(*----------------------------------------------------------------------------------------------------------------------------------------*)
(*Invoke Large Type Services Stand (Pnuematic I/O)*)
(*----------------------------------------------------------------------------------------------------------------------------------------*)
	(*Input Data*)
	SS01.Prev_EcatNode_Present:= NOT IS01.EK1100_NotPresent; (*Ensure Previous Node Exists to determine Ecat Cable Break of this Devices Input Cable*)
	SS01.Output_Req.0:= All_Estops_OK AND GTAC_CONFIG.Option_Air1; (*air valve 1*)
	SS01.Output_Req.1:= All_Estops_OK AND GTAC_CONFIG.Option_Air1; (*air valve 2*)
	SS01.Output_REQ.2:= RollDoor01.DoorClose_CMD;
	SS01.Output_REQ.3:= RollDoor01.DoorOpen_CMD;
	SS01.Output_REQ.4:= FALSE;
	SS01.Output_REQ.5:= FALSE;
	SS01.Output_REQ.6:= FALSE;
	SS01.Output_REQ.7:= FALSE;
	SS01.FB_In.Option_EP9214_Count:= GTAC_CONFIG.Option_EP9214_Count;
	(*Call Actual Function*)
	SS01();
	(*Output Data*)
	Out_To_ICxx.SS[1].Discrete_Image:= SS01.Discrete_Image;
	Out_To_ICxx.SS[1].ECAT_Cable_Breaks:= SS01.EcatSlave_Cable_Breaks;

	(*Input Data*)
	(*SS02.Prev_EcatNode_Present:= NOT SS01.EP1008_NotPresent; (*Ensure Previous Node Exists to determine Ecat Cable Break of this Devices Input Cable*)
	SS02.Output_Req.0:= All_Estops_OK AND GTAC_CONFIG.Option_Air2; (*air valve 1*)
	SS02.Output_Req.1:= All_Estops_OK AND GTAC_CONFIG.Option_Air2; (*air valve 2*)
	SS02.Output_REQ.2:= FALSE;
	SS02.Output_REQ.3:= FALSE;
	SS02.Output_REQ.4:= FALSE;
	SS02.Output_REQ.5:= FALSE;
	SS02.Output_REQ.6:= FALSE;
	SS02.Output_REQ.7:= FALSE;
	(*Call Actual Function*)
	SS02();
	(*Output Data*)
	Out_To_ICxx.SS[2].Discrete_Image:= SS02.Discrete_Image;
	Out_To_ICxx.SS[2].ECAT_Cable_Breaks:= SS02.EcatSlave_Cable_Breaks;*)


(*----------------------------------------------------------------------------------------------------------------------------------------*)
(* Invoke Enabling Swtich Plates*)
(*----------------------------------------------------------------------------------------------------------------------------------------*)
	(*Input Data*)
	ESW01.Prev_EcatNode_Present:= NOT MAIN.R3.EL6695_PortC_MissingLink; (*Ensure Previous Node Exists to determine Ecat Cable Break of this Devices Input Cable*)
	(*Call Actual Function*)
	ESW01();
	(*Output Data*)
	Out_To_ICxx.ESW[1].Discrete_Image:= ESW01.Discrete_Image;
	Out_To_ICxx.ESW[1].ECAT_Cable_Breaks:= ESW01.EcatSlave_Cable_Breaks;
	
	(*Input Data*)
	ESW02.Prev_EcatNode_Present:= NOT MAIN.IC03.EK1100_NotPresent; (*Ensure Previous Node Exists to determine Ecat Cable Break of this Devices Input Cable*)
	(*Call Actual Function*)
	ESW02();
	(*Output Data*)
	Out_To_ICxx.ESW[2].Discrete_Image:= ESW02.Discrete_Image;
	Out_To_ICxx.ESW[2].ECAT_Cable_Breaks:= ESW02.EcatSlave_Cable_Breaks;

	(*Input Data*)
	ESW03.Prev_EcatNode_Present:= NOT MAIN.IC02.EK1100_NotPresent; (*Ensure Previous Node Exists to determine Ecat Cable Break of this Devices Input Cable*)
	(*Call Actual Function*)
	ESW03();
	(*Output Data*)
	Out_To_ICxx.ESW[3].Discrete_Image:= ESW03.Discrete_Image;
	Out_To_ICxx.ESW[3].ECAT_Cable_Breaks:= ESW03.EcatSlave_Cable_Breaks;

(*----------------------------------------------------------------------------------------------------------------------------------------*)
(*Invoke EOAT FBs and Subordinate Fixtures*)
(*----------------------------------------------------------------------------------------------------------------------------------------*)
	(*EOATs Action*)
	EOATs();

(*----------------------------------------------------------------------------------------------------------------------------------------*)
(*Invoke IC FBs and Subordinate Fixtures*)
(*----------------------------------------------------------------------------------------------------------------------------------------*)
	(*ICs Action*)
	ICs();
	
(*----------------------------------------------------------------------------------------------------------------------------------------*)
(*Invoke Product Tracking Action*)
(*----------------------------------------------------------------------------------------------------------------------------------------*)
	(*Product Tracking Action*)
	Product_Tracking();

(*-------------------------------------------------------------------------------------------------------------------------------------*)
(*Invoke Robot FBs*)
(*-------------------------------------------------------------------------------------------------------------------------------------*)
	(*Robots Action*)
	Robots();

	
(*-------------------------------------------------------------------------------------------------------------------------------------*)
(*-------------------------------------------------------------------------------------------------------------------------------------*)
(*---------------------------------------------------- End of MAIN---------------------------------------------------------------------*)
(*-------------------------------------------------------------------------------------------------------------------------------------*)
(*-------------------------------------------------------------------------------------------------------------------------------------*)

ACTION EOATs:



	(*R04 - EOAT 04*)
		EOAT04(

			Enable_Motion:= R4.Servos_Are_On,
			Dry_Cycle:= GTAC_CONFIG.Dry_Cycle_Enabled,
			Robot_WorkingOK:= ((R4.Task_ID_Ack=PickUP_Fix01) OR (R4.Task_ID_Ack=Work_PED01)) AND R4.Operating,

			(*Set Configuration Data Here*)
			ID:= 4,							(*Set EOAT ID*)
			NodeLayout:= Main.ECAT_Master.EOATNodeLayout[4],	(*Pass in Assembled Node layout for UI*)
			Input_Node_Count:= 5,				(*Set Expected Input Node Count(Current Limit is 9*)
			VB_Node_Count:= 1,				(*Set Expected Input Node Count(Current Limit is 3*)
	
			(*Input Data*)
			(*Use Command All Sensors if your gripper has common part for the entire gripper.*)
			(*Use Command Sensors Group1/Group 2 if your gripper has multiple parts for the entire gripper. EX: LH and RH part*)
			CMD_CheckAllSensors_OFF:= FALSE, 
			CMD_CheckSensorsOFF_Grp1:= R4.EOAT_Req.0, (*129*) (*Sensors 1-2*)
			CMD_CheckSensorsOFF_Grp2:= R4.EOAT_Req.2, (*131*) (*Sensors 3-4*)
			CMD_CheckSensorsOFF_Grp3:= FALSE,
			CMD_CheckSensorsOFF_Grp4:= FALSE,
			CMD_CheckSensorsOFF_Grp5:= FALSE,

			CMD_CheckAllSensors_ON:= FALSE,
			CMD_CheckSensorsON_Grp1:= R4.EOAT_Req.1, (*130*) (*Sensors 1-2*)
			CMD_CheckSensorsON_Grp2:= R4.EOAT_Req.3, (*132*) (*Sensors 3-4*)
			CMD_CheckSensorsON_Grp3:= FALSE,
			CMD_CheckSensorsON_Grp4:= FALSE,
			CMD_CheckSensorsON_Grp5:= FALSE,

			(*Use Command Tool to Work/HOME if your gripper has common part for the entire gripper.*)
			(*Use Clamps Groups if your gripper has a LH/RH part for the gripper.*)
			CMD_Tool_To_WORK:= FALSE,
			CMD_CylToWORK_Grp1:= R4.EOAT_Req.4, (*133*) (*Clamps 1-4*)
			CMD_CylToWORK_Grp2:= R4.EOAT_Req.6, (*135*) (*Clamps 5-8*)
			CMD_CylToWORK_Grp3:= R4.EOAT_Req.8, (*137*) (*Pins 1-2*)
			CMD_CylToWORK_Grp4:= R4.EOAT_Req.10, (*139*) (*Pins 3-4*)
			CMD_CylToWORK_Grp5:= FALSE,

			CMD_Tool_To_HOME:= FALSE,
			CMD_CylToHOME_Grp1:= R4.EOAT_Req.5, (*134*) (*Clamps 1-4*)
			CMD_CylToHOME_Grp2:= R4.EOAT_Req.7, (*136*) (*Clamps 5-8*)
			CMD_CylToHOME_Grp3:= R4.EOAT_Req.9, (*138*) (*Pins 1-2*)
			CMD_CylToHOME_Grp4:= R4.EOAT_Req.11, (*140*) (*Pins 3-4*)
			CMD_CylToHOME_Grp5:= FALSE
			);
		(*Output Data*)
		Out_To_ICxx.EOAT04_Discrete_Image:= EOAT04.Discrete_Image;
		Out_To_ICxx.ProductReport[34]:= EOAT04_1_ProductData_Pers; 	(*Transfer Product Data to UI*)
		Out_To_ICxx.ProductReport[35]:= EOAT04_2_ProductData_Pers; 	(*Transfer Product Data to UI*)

		(*Output Data - Send ACKs bak to Robot*)
		(*Sensor ACKs*)
		R4.FB_In.EOATReq_Ack.0:= EOAT04.EOAT_Part1_Empty;	(*129*) //R4.EOAT_Req.0 AND DEBUG - removed to make more automated. delete if tested good
		R4.FB_In.EOATReq_Ack.1:= EOAT04.Part1_In_EOAT;		(*130*) //R4.EOAT_Req.1 AND DEBUG
		R4.FB_In.EOATReq_Ack.2:= EOAT04.EOAT_Part2_Empty;	(*131*) //R4.EOAT_Req.2 AND DEBUG 
		R4.FB_In.EOATReq_Ack.3:= EOAT04.Part2_In_EOAT;		(*132*) //R4.EOAT_Req.3 AND DEBUG
		
		(*CLAMP ACKs*)
		R4.FB_In.EOATReq_Ack.4:= R4.EOAT_Req.4 AND EOAT04.ACK_CylAtWORK_Grp1;	(*133*)
		R4.FB_In.EOATReq_Ack.5:= R4.EOAT_Req.5 AND EOAT04.ACK_CylAtHOME_Grp1;	(*134*)		
		R4.FB_In.EOATReq_Ack.6:= R4.EOAT_Req.6 AND EOAT04.ACK_CylAtWORK_Grp2;	(*135*)
		R4.FB_In.EOATReq_Ack.7:= R4.EOAT_Req.7 AND EOAT04.ACK_CylAtHOME_Grp2;	(*136*)
		
		(*Pin ACKs*)
		R4.FB_In.EOATReq_Ack.8:= R4.EOAT_Req.8 AND EOAT04.ACK_CylAtWORK_Grp3;	(*137*)
		R4.FB_In.EOATReq_Ack.9:= R4.EOAT_Req.9 AND EOAT04.ACK_CylAtHOME_Grp3;	(*138*)		
		R4.FB_In.EOATReq_Ack.10:= R4.EOAT_Req.10 AND EOAT04.ACK_CylAtWORK_Grp4;	(*139*)
		R4.FB_In.EOATReq_Ack.11:= R4.EOAT_Req.11 AND EOAT04.ACK_CylAtHOME_Grp4;	(*140*)

	(*Additional EOAT can be added here. Up to 30*)
	(*Please update the faults if you add additional EOAT*)
END_ACTION

ACTION ICs:



	(*Industrial Controller 01*)
	(*Input Data*)
	IC01.FB_In.Safety_RST:=SAFETY_RESET;
	IC01.FB_In.Enable_Motion:= All_Estops_OK AND All_SafetyGates_OK;
	IC01.FB_In.Estops_OK:= All_Estops_OK;
	IC01.FB_In.Safety_Gates_Ok:= All_SafetyGates_OK;
	IC01.FB_In.CoE_Read_Trigger:= (GTAC_CONFIG.Option_IC_Count>=1) AND Pulse_CoERead;	(*Global Interval of CoE Reads*)
	IC01.FB_In.Ecat_Master_AmsNetID:= MAIN.ECAT_Master.AmsID;
	IC01.FB_In.Prev_EcatNode_Present:= TRUE; 												(*Ensure Previous Node Exists to determine Ecat Cable Break of this Devices Input Cable*)
	IC01.FB_In.Output_Req1:= In_From_ICxx.LockSGK1;
	IC01.Turntable_Type:= TRUE;	(*Debug - Set to true if using a turntable. this will change the status light based on table position. set to false if no turntable.*)
	IC01.Op1_At_Operator:= Fix01.TurntableB_At_Robot OR (MAIN.R1.Task_ID_Ack=Sweep_Fix01) OR (MAIN.R2.Task_ID_Ack=Sweep_Fix01) OR (MAIN.R1.Task_ID_Ack=Sweep_Fix02) OR (MAIN.R2.Task_ID_Ack=Sweep_Fix02);
	IC01.Op2_At_Operator:= Fix01.TurntableA_At_Robot OR (MAIN.R1.Task_ID_Ack=Sweep_Fix01) OR (MAIN.R2.Task_ID_Ack=Sweep_Fix01) OR (MAIN.R1.Task_ID_Ack=Sweep_Fix02) OR (MAIN.R2.Task_ID_Ack=Sweep_Fix02);
	IC01.FB_In.OP1_Green_LampReq:= Fix01.Ready_To_Load;
	IC01.FB_In.OP2_Green_LampReq:= Fix03.Ready_To_Load;
	IC01.FB_In.OP1_Yellow_LampReq:= TRUE;
	IC01.FB_In.OP2_Yellow_LampReq:= TRUE;
	IC01.FB_In.OP1_Red_LampReq:= Fix01.Red_Lamp_Req OR Faults.System_Major_Fault;
	IC01.FB_In.OP2_Red_LampReq:= Fix03.Red_Lamp_Req OR Faults.System_Major_Fault;
	IC01.OP1_LC_Clear:= IC01.OP1_HumanVertLC_Clear AND IC01.OP1_HumanHorizLC_Clear AND IC01.OP1_RobotVertLC_Clear AND IC01.OP2_HumanVertLC_Clear AND IC01.OP2_HumanHorizLC_Clear;
	IC01.OP2_LC_Clear:= IC01.OP1_HumanVertLC_Clear AND IC01.OP1_HumanHorizLC_Clear AND IC01.OP1_RobotVertLC_Clear AND IC01.OP2_HumanVertLC_Clear AND IC01.OP2_HumanHorizLC_Clear;
	(*Call FUNCTION*)
	IC01();
	(*Output IC Data to All ICs*)
	Out_To_ICxx.IC[1].Discrete_Image:= IC01.Discrete_Image;
	Out_To_ICxx.IC[1].ECAT_Cable_Breaks:= IC01.ECatSlave_Cable_Breaks;
	Out_To_ICxx.IC01OP1_LCHVR:= IC01.OP1_HumanVertLC_Clear;
	Out_To_ICxx.IC01OP1_LCHHR:= IC01.OP1_HumanHorizLC_Clear;
	Out_To_ICxx.IC01OP1_LCRVR:= IC01.OP1_RobotVertLC_Clear; (*DEBUG - ADD OR REMOVE TO OTHER LIGHT CURTAINS. BYPASSES INDICATOR ON UI*)
	Out_To_ICxx.IC01OP2_LCHVR:= IC01.OP2_HumanVertLC_Clear;
	Out_To_ICxx.IC01OP2_LCHHR:= IC01.OP2_HumanHorizLC_Clear;
	Out_To_ICxx.IC01OP2_LCRVR:= IC01.OP2_RobotVertLC_Clear;
	
		(*OP1*)
			(*Fixture 01*)
			(*Input Data*)
			Fix01.Enable_Motion:= IC01.OP1_Enable_Motion;
			Fix01.Discrete_In:= In_From_ICxx.Fix01_Discrete_In;
			Fix01.Discrete_In.ModelData:= In_From_ICxx.Fix01_Discrete_In.ModelData;
			Fix01.NodeLayout:= Main.ECAT_Master.FixNodeLayout[1];				(*Pass in Assembled Node layout for UI*)
			Fix01.Discrete_In.Input_Node_Count:= 29;								(*Overridden for now, later version will map from UI read config sheet*)
			Fix01.Discrete_In.VB_Node_Count:= 2;								(*Overridden for now, later version will map from UI read config sheet*)
			Fix01.Discrete_In.Output_Node_Count:= 0;								(*Overridden for now, later version will map from UI read config sheet*)
			Fix01.Discrete_In.Water_Stand_Count:= 0;							(*Overridden for now, later version will map from UI read config sheet*)
			Fix01.Dry_Cycle:= GTAC_CONFIG.Dry_Cycle_Enabled OR GTAC_CONFIG.Local_DryCycle_Enables.1;
			Fix01.Cell_In_Services:= Cell_Services_Prog.Service_Call_ForAllRobots OR In_From_ICxx.Cycle_Hold;
			Fix01.Flash_Rate:= Pulse_1S;

			(*Call FUNCTION*)
			Fix01();
			(*Output Data*)
			Out_To_ICxx.Fix01_Discrete_Image:= Fix01.Discrete_Image;

		
			(*Fixture 02*)
			(*Input Data*)
			Fix02.Enable_Motion:= IC01.OP2_Enable_Motion;
			Fix02.Discrete_In:= In_From_ICxx.Fix02_Discrete_In;
			Fix02.Discrete_In.ModelData:= In_From_ICxx.Fix02_Discrete_In.ModelData;
			Fix02.NodeLayout:= Main.ECAT_Master.FixNodeLayout[2];				(*Pass in Assembled Node layout for UI*)
			Fix02.Discrete_In.Input_Node_Count:= 29;								(*Overridden for now, later version will map from UI read config sheet*)
			Fix02.Discrete_In.VB_Node_Count:= 2;								(*Overridden for now, later version will map from UI read config sheet*)
			Fix02.Discrete_In.Output_Node_Count:= 0;								(*Overridden for now, later version will map from UI read config sheet*)
			Fix02.Discrete_In.Water_Stand_Count:= 0;								(*Overridden for now, later version will map from UI read config sheet*)
			Fix02.Dry_Cycle:= GTAC_CONFIG.Dry_Cycle_Enabled OR GTAC_CONFIG.Local_DryCycle_Enables.2;
			Fix02.Cell_In_Services:= Cell_Services_Prog.Service_Call_ForAllRobots OR In_From_ICxx.Cycle_Hold;
			Fix02.Flash_Rate:= Pulse_1S;
			(*Call FUNCTION*)
			Fix02();
			(*Output Data*)
			Out_To_ICxx.Fix02_Discrete_Image:= Fix02.Discrete_Image;

	(*Industrial Controller 02*)
	(*Input Data*)
	IC02.FB_In.Safety_RST:=SAFETY_RESET;
	IC02.FB_In.Enable_Motion:= All_Estops_OK AND All_SafetyGates_OK;
	IC02.FB_In.Estops_OK:= All_Estops_OK;
	IC02.FB_In.Safety_Gates_Ok:= All_SafetyGates_OK;
	IC02.FB_In.CoE_Read_Trigger:= (GTAC_CONFIG.Option_IC_Count>=2) AND Pulse_CoERead;	(*Global Interval of CoE Reads*)
	IC02.FB_In.Ecat_Master_AmsNetID:= MAIN.ECAT_Master.AmsID;
	IC02.FB_In.Prev_EcatNode_Present:= NOT MAIN.MD02.EP2624_PortB_MissingLink ; 						(*Ensure Previous Node Exists to determine Ecat Cable Break of this Devices Input Cable*)
	IC02.FB_In.Output_Req1:= In_From_ICxx.LockSGK1 OR In_From_ICxx.LockSGK2;
	IC02.Turntable_Type:= TRUE;	(*Debug - Set to true if using a turntable. this will change the status light based on table position. set to false if no turntable.*)
	IC02.Op1_At_Operator:= Fix03.TurntableB_At_Robot OR (MAIN.R3.Task_ID_Ack=Sweep_Fix03) OR (MAIN.R4.Task_ID_Ack=Sweep_Fix03) OR (MAIN.R3.Task_ID_Ack=Sweep_Fix04) OR (MAIN.R4.Task_ID_Ack=Sweep_Fix04); (*debug - change robot*)
	IC02.Op2_At_Operator:= Fix03.TurntableA_At_Robot OR (MAIN.R3.Task_ID_Ack=Sweep_Fix03) OR (MAIN.R4.Task_ID_Ack=Sweep_Fix03) OR (MAIN.R3.Task_ID_Ack=Sweep_Fix04) OR (MAIN.R4.Task_ID_Ack=Sweep_Fix04); (*debug - change robot*)
	IC02.FB_In.OP1_Green_LampReq:= Fix03.Ready_To_Load;
	IC02.FB_In.OP2_Green_LampReq:= Fix04.Ready_To_Load;
	IC02.FB_In.OP1_Yellow_LampReq:= TRUE;
	IC02.FB_In.OP2_Yellow_LampReq:= TRUE;
	IC02.FB_In.OP1_Red_LampReq:= Fix03.Red_Lamp_Req OR Faults.System_Major_Fault;
	IC02.FB_In.OP2_Red_LampReq:= Fix04.Red_Lamp_Req OR Faults.System_Major_Fault;
	IC02.OP1_LC_Clear:= IC02.OP1_HumanVertLC_Clear AND IC02.OP1_HumanHorizLC_Clear AND IC02.OP1_RobotVertLC_Clear AND IC02.OP2_HumanVertLC_Clear AND IC02.OP2_HumanHorizLC_Clear;
	IC02.OP2_LC_Clear:= IC02.OP1_HumanVertLC_Clear AND IC02.OP1_HumanHorizLC_Clear AND IC02.OP1_RobotVertLC_Clear AND IC02.OP2_HumanVertLC_Clear AND IC02.OP2_HumanHorizLC_Clear;
	(*Call FUNCTION*)
	IC02();
	(*Output IC Data to all ICs*)
	Out_To_ICxx.IC[2].Discrete_Image:= IC02.Discrete_Image;
	Out_To_ICxx.IC[2].ECAT_Cable_Breaks:= IC02.ECatSlave_Cable_Breaks;
	Out_To_ICxx.IC02OP1_LCHVR:= IC02.OP1_HumanVertLC_Clear;
	Out_To_ICxx.IC02OP1_LCHHR:= IC02.OP1_HumanHorizLC_Clear;
	Out_To_ICxx.IC02OP1_LCRVR:= IC02.OP1_RobotVertLC_Clear;
	Out_To_ICxx.IC02OP2_LCHVR:= IC02.OP2_HumanVertLC_Clear;
	Out_To_ICxx.IC02OP2_LCHHR:= IC02.OP2_HumanHorizLC_Clear;
	Out_To_ICxx.IC02OP2_LCRVR:= IC02.OP2_RobotVertLC_Clear;

		(*OP1*)
			(*Fixture 03*)
			(*Input Data*)
			Fix03.Enable_Motion:= IC02.OP1_Enable_Motion;
			Fix03.Discrete_In:= In_From_ICxx.Fix03_Discrete_In;
			(*Perform Look ahead for Model data depending on line loading*)
			
				(*Valid part For this Fix in EOAT04_1, so use EOAT_1 model*)
				IF ((EOAT04.Part1_In_EOAT AND NOT Fix03.Load_Complete) OR Fix03.Repo_REQS.0) AND Fix03.Part_InEOAT04_1_ReadyforThisFix 
					THEN
					Fix03.Discrete_In.ModelData:= EOAT04_1_ProductData_Pers.Product_Model_ID;
	
				(*Valid part For this Fix in EOAT04_2, so use EOAT_2 model*)
				ELSIF ((EOAT04.Part2_In_EOAT AND NOT Fix03.Load_Complete) OR Fix03.Repo_REQS.0) AND Fix03.Part_InEOAT04_2_ReadyforThisFix
					THEN
					Fix03.Discrete_In.ModelData:= EOAT04_2_ProductData_Pers.Product_Model_ID;
	
				(*No valid part in EOAT04, but valid part in Fix101, so use Fix101 model*)
				ELSIF (((NOT Fix03.Load_Complete OR Fix03.Unload_Complete) AND Fix101.Load_Complete) OR (MAIN.R4.Task_ID_Ack = PickUp_Fix101)) AND 
						NOT Fix03.Part_InEOAT04_1_ReadyforThisFix AND NOT Fix03.Part_InEOAT04_2_ReadyforThisFix AND (MAIN.R4.Task_ID_Ack <> DropOff_Fix03)
					THEN
					Fix03.Discrete_In.ModelData:= Fix101_ProductData_Pers.Product_Model_ID;
	
				(*No valid part in Fix101 but valid part in EOAT04_1 for Fix101, so use EOAT04_1 model*)
				ELSIF NOT Fix03.Load_Complete AND NOT Fix101.Load_Complete AND (MAIN.R4.Task_ID_Ack <> PickUp_Fix101) AND Fix101.Part_InEOAT04_1_ReadyforThisFix 
					THEN
					Fix03.Discrete_In.ModelData:= EOAT04_1_ProductData_Pers.Product_Model_ID;
	
				(*No valid part in Fix101 but valid part in EOAT04_2 for Fix101, so use EOAT04_1 model*)
				ELSIF NOT Fix03.Load_Complete AND NOT Fix101.Load_Complete AND (MAIN.R4.Task_ID_Ack <> PickUp_Fix101) AND Fix101.Part_InEOAT04_2_ReadyforThisFix 
					THEN
					Fix03.Discrete_In.ModelData:= EOAT04_2_ProductData_Pers.Product_Model_ID;
	
				(*No valid part in Fix101, no Valid part in EOAT04 but model in Fix01 / 02 AND Fix03 empty*)
				ELSIF (NOT Fix03.Load_Complete OR Fix03.Unload_Complete) AND NOT Fix101.Load_Complete AND (MAIN.R4.Task_ID_Ack <> PickUp_Fix101) AND 
							NOT Fix101.Part_InEOAT04_1_ReadyforThisFix AND NOT Fix101.Part_InEOAT04_2_ReadyforThisFix AND 
							NOT Fix03.Part_InEOAT04_1_ReadyforThisFix AND NOT Fix03.Part_InEOAT04_2_ReadyforThisFix 
					THEN
					(*Fix01 Faces Weld Robots*)
					IF (Out_To_ICxx.TT01_Location_Index = 1) AND NOT Fix01.All_Sensors_Off AND (MAIN.R4.Task_ID_Ack <> DropOff_Fix03)
						THEN
						Fix03.Discrete_In.ModelData:= Fix01_ProductData_Pers.Product_Model_ID;
					(*Fix02 Faces Weld Robots*)	
					ELSIF (Out_To_ICxx.TT01_Location_Index = 2) AND NOT Fix02.All_Sensors_Off AND (MAIN.R4.Task_ID_Ack <> DropOff_Fix03)
						THEN	
						Fix03.Discrete_In.ModelData:= Fix02_ProductData_Pers.Product_Model_ID;
					ELSIF
						((Out_To_ICxx.TT01_Location_Index = 1) OR (Out_To_ICxx.TT01_Location_Index = 2)) AND Fix01.All_Sensors_Off AND Fix02.All_Sensors_Off
						THEN
						Fix03.Discrete_In.ModelData:= Fix01_ProductData_Pers.Product_Model_ID;
					END_IF;
				END_IF;
(*
				(*FINALLY, if part has been loaded onto this Fix, so use local model data *)
				ELSIF   (Fix03.Load_Complete AND (MAIN.R4.Task_ID_Ack <> DropOff_Fix03)) OR Fix03.Repo_REQS.0
					THEN
						test1:= TRUE;
						Fix03.Discrete_In.ModelData:= Fix03_ProductData_Pers.Product_Model_ID;
				END_IF;  DEBUG - this partially works... not a clue why  - rj*)
				
				(*FINALLY, if part has been loaded onto this Fix, so use local model data *)
				IF   (Fix03.Load_Complete OR Fix03.Repo_REQS.0) AND ((MAIN.R4.Task_ID_Ack <> DropOff_Fix03) OR Fix03.Load_Robots_Complete1)
					 AND NOT Fix03.Unload_Complete
					THEN
						test1:= TRUE;
						Fix03.Discrete_In.ModelData:= Fix03_ProductData_Pers.Product_Model_ID;
				END_IF;
				
			Fix03.NodeLayout:= Main.ECAT_Master.FixNodeLayout[3];				(*Pass in Assembled Node layout for UI*)
			Fix03.Discrete_In.Input_Node_Count:= 21;								(*Overridden for now, later version will map from UI read config sheet*)
			Fix03.Discrete_In.VB_Node_Count:= 1;								(*Overridden for now, later version will map from UI read config sheet*)
			Fix03.Discrete_In.Output_Node_Count:= 0;								(*Overridden for now, later version will map from UI read config sheet*)
			Fix03.Discrete_In.Water_Stand_Count:= 0;								(*Overridden for now, later version will map from UI read config sheet*)
			Fix03.Dry_Cycle:= GTAC_CONFIG.Dry_Cycle_Enabled OR GTAC_CONFIG.Local_DryCycle_Enables.3;
			Fix03.Cell_In_Services:= Cell_Services_Prog.Service_Call_ForAllRobots OR In_From_ICxx.Cycle_Hold;
			Fix03.Flash_Rate:= Pulse_1S;
			(*Call FUNCTION*)
			Fix03();
			(*Output Data*)
			Out_To_ICxx.Fix03_Discrete_Image:= Fix03.Discrete_Image;


		(*OP2*)
			(*Fixture 04*)
			(*Input Data*)
			Fix04.Enable_Motion:= IC02.OP2_Enable_Motion;
			Fix04.Discrete_In:= In_From_ICxx.Fix04_Discrete_In;
			
				(*Perform Look ahead for Model data depending on line loading*)
			
				(*Valid part For this Fix in EOAT04_1, so use EOAT_1 model*)
				IF ((EOAT04.Part1_In_EOAT AND NOT Fix04.Load_Complete) OR Fix04.Repo_REQS.0) AND Fix04.Part_InEOAT04_1_ReadyforThisFix
					THEN
					Fix04.Discrete_In.ModelData:= EOAT04_1_ProductData_Pers.Product_Model_ID;
	
				(*Valid part For this Fix in EOAT04_2, so use EOAT_2 model*)
				ELSIF ((EOAT04.Part2_In_EOAT AND NOT Fix04.Load_Complete) OR Fix04.Repo_REQS.0) AND Fix04.Part_InEOAT04_2_ReadyforThisFix
					THEN
					Fix04.Discrete_In.ModelData:= EOAT04_2_ProductData_Pers.Product_Model_ID;
	
				(*No valid part in EOAT04, but valid part in Fix101, so use Fix101 model*)
				ELSIF NOT Fix04.Load_Complete AND Fix101.Load_Complete OR (MAIN.R4.Task_ID_Ack = PickUp_Fix101) AND 
						NOT Fix04.Part_InEOAT04_1_ReadyforThisFix AND NOT Fix04.Part_InEOAT04_2_ReadyforThisFix
					THEN
					Fix04.Discrete_In.ModelData:= Fix101_ProductData_Pers.Product_Model_ID;
	
				(*No valid part in Fix101 but valid part in EOAT04_1 for Fix101, so use EOAT04_1 model*)
				ELSIF NOT Fix04.Load_Complete AND NOT Fix101.Load_Complete AND (MAIN.R4.Task_ID_Ack <> PickUp_Fix101) AND Fix101.Part_InEOAT04_1_ReadyforThisFix
					THEN
					Fix04.Discrete_In.ModelData:= EOAT04_1_ProductData_Pers.Product_Model_ID;
	
				(*No valid part in Fix101 but valid part in EOAT04_2 for Fix101, so use EOAT04_1 model*)
				ELSIF NOT Fix04.Load_Complete AND NOT Fix101.Load_Complete AND (MAIN.R4.Task_ID_Ack <> PickUp_Fix101) AND Fix101.Part_InEOAT04_2_ReadyforThisFix
					THEN
					Fix04.Discrete_In.ModelData:= EOAT04_2_ProductData_Pers.Product_Model_ID;
	
				(*No valid part in Fix101, no Valid part in EOAT04 but model in Fix01 / 02*)
				ELSIF NOT Fix04.Load_Complete and NOT Fix101.Load_Complete AND (MAIN.R4.Task_ID_Ack <> PickUp_Fix101) AND 
							NOT Fix101.Part_InEOAT04_1_ReadyforThisFix AND NOT Fix101.Part_InEOAT04_2_ReadyforThisFix AND 
							NOT Fix04.Part_InEOAT04_1_ReadyforThisFix AND NOT Fix04.Part_InEOAT04_2_ReadyforThisFix
					THEN
					(*Fix01 Faces Weld Robots*)
					IF (Out_To_ICxx.TT01_Location_Index = 1)
						THEN
						Fix04.Discrete_In.ModelData:= Fix01_ProductData_Pers.Product_Model_ID;
					(*Fix02 Faces Weld Robots*)	
					ELSIF (Out_To_ICxx.TT01_Location_Index = 2)
						THEN	
						Fix04.Discrete_In.ModelData:= Fix02_ProductData_Pers.Product_Model_ID;
					END_IF;
	
				(*FINALLY, if part has been loaded onto this Fix, so use local model data*)
				ELSIF (Fix04.Load_Complete OR Fix04.Repo_REQS.1) AND (MAIN.R4.Task_ID_Ack <> DropOff_Fix04)
					THEN
					Fix04.Discrete_In.ModelData:= Fix04_ProductData_Pers.Product_Model_ID;
				END_IF;
				
			Fix04.NodeLayout:= Main.ECAT_Master.FixNodeLayout[4];				(*Pass in Assembled Node layout for UI*)
			Fix04.Discrete_In.Input_Node_Count:= 22;								(*Overridden for now, later version will map from UI read config sheet*)
			Fix04.Discrete_In.VB_Node_Count:= 1;								(*Overridden for now, later version will map from UI read config sheet*)
			Fix04.Discrete_In.Output_Node_Count:= 0;								(*Overridden for now, later version will map from UI read config sheet*)
			Fix04.Discrete_In.Water_Stand_Count:= 0;								(*Overridden for now, later version will map from UI read config sheet*)
			Fix04.Dry_Cycle:= GTAC_CONFIG.Dry_Cycle_Enabled OR GTAC_CONFIG.Local_DryCycle_Enables.4;
			Fix04.Cell_In_Services:= Cell_Services_Prog.Service_Call_ForAllRobots OR In_From_ICxx.Cycle_Hold;
			Fix04.Flash_Rate:= Pulse_1S;
			(*Call FUNCTION*)
			Fix04();
			(*Output Data*)
			Out_To_ICxx.Fix04_Discrete_Image:= Fix04.Discrete_Image;

	(*Industrial Controller 03*)
	(*Input Data*)
	IC03.FB_In.Safety_RST:=SAFETY_RESET;
	IC03.FB_In.Enable_Motion:= All_Estops_OK AND All_SafetyGates_OK;
	IC03.FB_In.Estops_OK:= All_Estops_OK;
	IC03.FB_In.Safety_Gates_Ok:= All_SafetyGates_OK;
	IC03.FB_In.CoE_Read_Trigger:= (GTAC_CONFIG.Option_IC_Count>=3) AND Pulse_CoERead;	(*Global Interval of CoE Reads*)
	IC03.FB_In.Ecat_Master_AmsNetID:= MAIN.ECAT_Master.AmsID;
	IC03.FB_In.Prev_EcatNode_Present:= NOT MAIN.R11.EL6695_PortC_MissingLink; 						(*Ensure Previous Node Exists to determine Ecat Cable Break of this Devices Input Cable*)
	IC03.FB_In.Output_Req1:= In_From_ICxx.LockSGK1;
	IC03.Turntable_Type:= FALSE;	(*Debug - Set to true if using a turntable. this will change the status light based on table position. set to false if no turntable.*)
	IC03.Op1_At_Operator:= Fix05.TurntableB_At_Robot OR (MAIN.R1.Task_ID_Ack=Sweep_Fix05) OR (MAIN.R2.Task_ID_Ack=Sweep_Fix05); (*debug - change robot*)
	IC03.Op2_At_Operator:= Fix05.TurntableA_At_Robot OR (MAIN.R1.Task_ID_Ack=Sweep_Fix05) OR (MAIN.R2.Task_ID_Ack=Sweep_Fix05); (*debug - change robot*)
	IC03.FB_In.OP1_Green_LampReq:= Fix05.Ready_To_Load;
	IC03.FB_In.OP2_Green_LampReq:= Fix05.Ready_To_Load;
	IC03.FB_In.OP1_Yellow_LampReq:= TRUE;
	IC03.FB_In.OP2_Yellow_LampReq:= TRUE;
	IC03.FB_In.OP1_Red_LampReq:= Fix05.Red_Lamp_Req OR Faults.System_Major_Fault;
	IC03.FB_In.OP2_Red_LampReq:= Fix06.Red_Lamp_Req OR Faults.System_Major_Fault;
	IC03.OP1_LC_Clear:= IC03.OP1_HumanVertLC_Clear AND IC03.OP1_HumanHorizLC_Clear (*AND IC03.OP1_RobotVertLC_Clear*);
	IC03.OP2_LC_Clear:= IC03.OP1_HumanVertLC_Clear AND IC03.OP1_HumanHorizLC_Clear (*IC03.OP2_HumanVertLC_Clear AND IC03.OP2_HumanHorizLC_Clear AND IC03.OP2_RobotVertLC_Clear*);
	(*Call FUNCTION*)
	IC03();
	(*Output IC Data to all ICs*)
	Out_To_ICxx.IC[3].Discrete_Image:= IC03.Discrete_Image;
	Out_To_ICxx.IC[3].ECAT_Cable_Breaks:= IC03.ECatSlave_Cable_Breaks;
	Out_To_ICxx.IC03OP1_LCHVR:= IC03.OP1_HumanVertLC_Clear;
	Out_To_ICxx.IC03OP1_LCHHR:= IC03.OP1_HumanHorizLC_Clear;
	Out_To_ICxx.IC03OP1_LCRVR:= IC03.OP1_RobotVertLC_Clear;
	Out_To_ICxx.IC03OP2_LCHVR:= IC03.OP2_HumanVertLC_Clear;
	Out_To_ICxx.IC03OP2_LCHHR:= IC03.OP2_HumanHorizLC_Clear;
	Out_To_ICxx.IC03OP2_LCRVR:= IC03.OP2_RobotVertLC_Clear;

		(*OP1*)
			(*Fixture 05*)
			(*Input Data*)
			Fix05.Enable_Motion:= IC03.OP1_Enable_Motion;
			Fix05.Discrete_In:= In_From_ICxx.Fix05_Discrete_In;
			Fix05.Discrete_In.ModelData:= In_From_ICxx.Fix05_Discrete_In.ModelData; (*DEBUG, will have to be finalized once Fix05 redesign is complete, blt*)
			Fix05.NodeLayout:= Main.ECAT_Master.FixNodeLayout[5];				(*Pass in Assembled Node layout for UI*)
			Fix05.Discrete_In.Input_Node_Count:= 4;								(*Overridden for now, later version will map from UI read config sheet*)
			Fix05.Discrete_In.VB_Node_Count:= 1;								(*Overridden for now, later version will map from UI read config sheet*)
			Fix05.Discrete_In.Output_Node_Count:= 0;								(*Overridden for now, later version will map from UI read config sheet*)
			Fix05.Discrete_In.Water_Stand_Count:= 0;								(*Overridden for now, later version will map from UI read config sheet*)
			Fix05.Dry_Cycle:= GTAC_CONFIG.Dry_Cycle_Enabled OR GTAC_CONFIG.Local_DryCycle_Enables.5;
			Fix05.Cell_In_Services:= Cell_Services_Prog.Service_Call_ForAllRobots OR In_From_ICxx.Cycle_Hold;
			Fix05.Flash_Rate:= Pulse_1S;
			(*Call FUNCTION*)
			Fix05();
			(*Output Data*)
			Out_To_ICxx.Fix05_Discrete_Image:= Fix05.Discrete_Image;


(*Internal Fixtures*)

			(*Fixture 101*)
			(*Input Data*)
			Fix101.Enable_Motion:= Main.Control_Power_ON;								(*ENSURE to bind proper Relay Bank*)
			Fix101.Discrete_In:= In_From_ICxx.Fix101_Discrete_In;
			IF ((EOAT04.Part1_In_EOAT AND NOT Fix101.Load_Complete) OR Fix101.Repo_REQS.0) AND Fix101.Part_InEOAT04_1_ReadyforThisFix
				THEN
				Fix101.Discrete_In.ModelData:= EOAT04_1_ProductData_Pers.Product_Model_ID;
			ELSIF (EOAT04_2_ProductData_Pers.Generic_PassFail_Notes[1] = '') // weld fix101 complete
					AND ((EOAT04.Part2_In_EOAT AND NOT Fix101.Load_Complete) OR Fix101.Repo_REQS.0) AND Fix101.Part_InEOAT04_2_ReadyforThisFix
				THEN
				Fix101.Discrete_In.ModelData:= EOAT04_2_ProductData_Pers.Product_Model_ID; 
			ELSIF (Fix101.Load_Complete OR Fix101.Repo_REQS.1) AND (MAIN.R4.Task_ID_Ack <> DropOff_Fix101) AND NOT Fix101.Unload_Complete
				THEN
				Fix101.Discrete_In.ModelData:= Fix101_ProductData_Pers.Product_Model_ID;
			ELSIF (Fix101.Unload_Complete AND Fix101.All_Sensors_Off AND NOT Main.R1.TT_at_Dropoff_Pos)
				THEN
				Fix101.Discrete_In.ModelData:= 1;
			ELSIF Fix101.All_Sensors_Off AND NOT Fix101.Part_InEOAT04_1_ReadyforThisFix AND NOT Fix101.Part_InEOAT04_2_ReadyforThisFix AND (MAIN.R4.Task_ID_Ack <> DropOff_Fix101)
				THEN 
				 IF 	(*Fix01 Faces Weld Robots*)
						Fix01.TurntableA_At_Robot AND (Fix01.Model_ID <> 0)
					THEN
						Fix101.Discrete_In.ModelData:= Fix01_ProductData_Pers.Product_Model_ID;
						(*Fix02 Faces Weld Robots*)	
				ELSIF 	Fix02.TurntableB_At_Robot AND (Fix02.Model_ID <> 0)
					THEN	
						Fix101.Discrete_In.ModelData:= Fix02_ProductData_Pers.Product_Model_ID;
				END_IF
			END_IF;
			Fix101.NodeLayout:= Main.ECAT_Master.FixNodeLayout[101];				(*Pass in Assembled Node layout for UI*)
			Fix101.Discrete_In.Input_Node_Count:= 4;								(*Overridden for now, later version will map from UI read config sheet*)
			Fix101.Discrete_In.VB_Node_Count:= 1;								(*Overridden for now, later version will map from UI read config sheet*)
			Fix101.Discrete_In.Output_Node_Count:= 0;								(*Overridden for now, later version will map from UI read config sheet*)
			Fix101.Discrete_In.Water_Stand_Count:= 0;								(*Overridden for now, later version will map from UI read config sheet*)
			Fix101.Dry_Cycle:= GTAC_CONFIG.Dry_Cycle_Enabled;
			Fix101.Cell_In_Services:= Cell_Services_Prog.Service_Call_ForAllRobots OR In_From_ICxx.Cycle_Hold;
			Fix101.Flash_Rate:= Pulse_1S;
			(*Call FUNCTION*)
			Fix101();
			(*Output Data*)
			Out_To_ICxx.Fix101_Discrete_Image:= Fix101.Discrete_Image;
			(*------------------------- Nutweld Based LVDT system -----------------------------------*)
				(*Debug example only, using Fix101 as Nutwelder host*)

				(*Nutweld LVDT1*)
				(*Input Data*).
				MAIN.NutWeld_LVDT[1].Model_ID:= Fix101.Model_ID;
				MAIN.NutWeld_LVDT[1].Option_InScaledValues:= TRUE;		(*Sets if the system is working in scalled or raw values*) 
				MAIN.NutWeld_LVDT[1].Save_LVDT_Conf:= In_From_ICxx.NutWeld_LVDT_Discrete_In[1].Save_LVDT_REQ; 
				MAIN.NutWeld_LVDT[1].Save_Nut_Conf:= In_From_ICxx.NutWeld_LVDT_Discrete_In[1].Save_Nut_REQ; 
				MAIN.NutWeld_LVDT[1].Raw_Transducer:= 0; (*DEBUG,  map analog card Channel here*) 
				MAIN.NutWeld_LVDT[1].Ready_For_Measurement:= MAIN.R1.In_From_ECAT.Robot_OUT[172]; (*DEBUG,  confirm this is the proper output for "Weld ServoGun at Force"*)
				MAIN.NutWeld_LVDT[1].Weld_Complete:= MAIN.R1.WCU1_Weld_Complete; 
				MAIN.NutWeld_LVDT[1].Reset_NutOK:= NOT MAIN.R1.In_AutoExt
												OR Fix101.Reset_All_Completes
												OR (Fix101.In_Manual AND Fix101.Discrete_In.Go_Home); 
				MAIN.NutWeld_LVDT[1].NutInput_UpperLimit[Fix101.Model_ID]:= In_From_ICxx_Pers.Config_NutWeld_LVDT[1].Nut_UpperLimit;
				MAIN.NutWeld_LVDT[1].NutInput_LowerLimit[Fix101.Model_ID]:= In_From_ICxx_Pers.Config_NutWeld_LVDT[1].Nut_LowerLimit;


				(*Call FB Instance*)
				MAIN.NutWeld_LVDT[1]();
				(*Output Data*)
				Out_To_ICxx.NutWeld_LVDT_Discrete_Image[1].LVDT_Saved_ACK:= MAIN.NutWeld_LVDT[1].LVDT_Saved;
				Out_To_ICxx.NutWeld_LVDT_Discrete_Image[1].LVDT_Value_Scaled:= MAIN.NutWeld_LVDT[1].NutPrev_Scaled;
				Out_To_ICxx.NutWeld_LVDT_Discrete_Image[1].LVDT_Value_Raw:= MAIN.NutWeld_LVDT[1].NutPrev_Raw;
				Out_To_ICxx.NutWeld_LVDT_Discrete_Image[1].LVDT_Nut_OK:= MAIN.NutWeld_LVDT[1].NutOK;
				
				(*----------------*)
				(*Outputs to Nutweld LVDT Discrete Image Area from Fix101 Pin13 (See Fix101.Cylinders.Pin13 example)*)
				Out_To_ICxx.NutWeld_LVDT_Discrete_Image[1].LVDT_Pin_RETD:= Fix101.Pin13RETD;
				Out_To_ICxx.NutWeld_LVDT_Discrete_Image[1].LVDT_Pin_ADVD:= Fix101.Pin13ADVD;
	
			(*-------------------------------------------------------------------------*)	
				
				
				
			(*Fixture 102*)
			(*Input Data*)
			Fix102.Enable_Motion:= Main.Control_Power_ON;								(*ENSURE to bind proper Relay Bank*)
			Fix102.Discrete_In:= In_From_ICxx.Fix102_Discrete_In;
			IF ((EOAT04.Part1_In_EOAT AND NOT Fix102.Load_Complete) OR Fix102.Repo_REQS.0) AND Fix102.Part_InEOAT04_1_ReadyforThisFix
				THEN
				Fix102.Discrete_In.ModelData:= EOAT04_1_ProductData_Pers.Product_Model_ID;
			ELSIF ((EOAT04.Part2_In_EOAT AND NOT Fix102.Load_Complete) OR Fix102.Repo_REQS.0) AND Fix102.Part_InEOAT04_2_ReadyforThisFix
				THEN
				Fix102.Discrete_In.ModelData:= EOAT04_2_ProductData_Pers.Product_Model_ID;
			ELSIF (Fix102.Load_Complete OR Fix102.Repo_REQS.0) AND (MAIN.R4.Task_ID_Ack <> DropOff_Fix102) AND NOT Fix102.Unload_Complete
				THEN
				Fix102.Discrete_In.ModelData:= Fix102_ProductData_Pers.Product_Model_ID;
				(*If nothing else is loaded, we need a model number to finish 102 sequance*)
			ELSIF (NOT Fix102.Load_Complete AND (NOT Fix03.Load_Complete OR NOT Fix04.Load_Complete) AND NOT Fix101.Load_Complete AND EOAT04.EOAT_Part1_Empty) 
				THEN
				Fix102.Discrete_In.ModelData:= Fix01_ProductData_Pers.Product_Model_ID;
			END_IF;
 			Fix102.NodeLayout:= Main.ECAT_Master.FixNodeLayout[102];				(*Pass in Assembled Node layout for UI*)
			Fix102.Discrete_In.Input_Node_Count:= 4;								(*Overridden for now, later version will map from UI read config sheet*)
			Fix102.Discrete_In.VB_Node_Count:= 1;								(*Overridden for now, later version will map from UI read config sheet*)
			Fix102.Discrete_In.Output_Node_Count:= 0;								(*Overridden for now, later version will map from UI read config sheet*)
			Fix102.Discrete_In.Water_Stand_Count:= 0;								(*Overridden for now, later version will map from UI read config sheet*)
			Fix102.Dry_Cycle:= GTAC_CONFIG.Dry_Cycle_Enabled;
			Fix102.Cell_In_Services:= Cell_Services_Prog.Service_Call_ForAllRobots OR In_From_ICxx.Cycle_Hold;
			Fix102.Flash_Rate:= Pulse_1S;
			(*Call FUNCTION*)
			Fix102();
			(*Output Data*)
			Out_To_ICxx.Fix102_Discrete_Image:= Fix102.Discrete_Image;


			(*Fixture 101*)
			(*Input Data*)
			Fix103.Enable_Motion:= Main.Control_Power_ON;							(*ENSURE to bind proper Relay Bank*)
			Fix103.Discrete_In:= In_From_ICxx.Fix103_Discrete_In;
			IF ((EOAT04.Part1_In_EOAT AND NOT Fix103.Load_Complete) OR Fix103.Repo_REQS.0) AND Fix103.Part_InEOAT04_1_ReadyforThisFix
				THEN
				Fix103.Discrete_In.ModelData:= EOAT04_1_ProductData_Pers.Product_Model_ID;
			ELSIF ((EOAT04.Part2_In_EOAT AND NOT Fix103.Load_Complete) OR Fix103.Repo_REQS.0) AND Fix103.Part_InEOAT04_2_ReadyforThisFix
				THEN
				Fix103.Discrete_In.ModelData:= EOAT04_2_ProductData_Pers.Product_Model_ID;
			ELSIF (Fix103.Load_Complete OR Fix103.Repo_REQS.1) AND (MAIN.R4.Task_ID_Ack <> DropOff_Fix103)
				THEN
				Fix103.Discrete_In.ModelData:= Fix103_ProductData_Pers.Product_Model_ID;
			END_IF;
 			Fix103.NodeLayout:= Main.ECAT_Master.FixNodeLayout[103];				(*Pass in Assembled Node layout for UI*)
			Fix103.Discrete_In.Input_Node_Count:= 2;								(*Overridden for now, later version will map from UI read config sheet*)
			Fix103.Discrete_In.VB_Node_Count:= 0;								(*Overridden for now, later version will map from UI read config sheet*)
			Fix103.Discrete_In.Output_Node_Count:= 0;								(*Overridden for now, later version will map from UI read config sheet*)
			Fix103.Discrete_In.Water_Stand_Count:= 0;								(*Overridden for now, later version will map from UI read config sheet*)
			Fix103.Dry_Cycle:= GTAC_CONFIG.Dry_Cycle_Enabled;
			Fix103.Cell_In_Services:= Cell_Services_Prog.Service_Call_ForAllRobots OR In_From_ICxx.Cycle_Hold;
			Fix103.Flash_Rate:= Pulse_1S;
			(*Call FUNCTION*)
			Fix103();
			(*Output Data*)
			Out_To_ICxx.Fix103_Discrete_Image:= Fix103.Discrete_Image;


			(*Fixture 101*)
			(*Input Data*)
			Fix104.Enable_Motion:= Main.Control_Power_ON;								(*ENSURE to bind proper Relay Bank*)
			Fix104.Discrete_In:= In_From_ICxx.Fix104_Discrete_In;
			IF ((EOAT04.Part1_In_EOAT AND NOT Fix104.Load_Complete) OR Fix104.Repo_REQS.0) AND Fix104.Part_InEOAT04_1_ReadyforThisFix
				THEN
				Fix104.Discrete_In.ModelData:= EOAT04_1_ProductData_Pers.Product_Model_ID;
			ELSIF ((EOAT04.Part2_In_EOAT AND NOT Fix104.Load_Complete) OR Fix104.Repo_REQS.0) AND Fix104.Part_InEOAT04_2_ReadyforThisFix
				THEN
				Fix104.Discrete_In.ModelData:= EOAT04_2_ProductData_Pers.Product_Model_ID;
			ELSIF (Fix104.Load_Complete OR Fix104.Repo_REQS.1) AND (MAIN.R4.Task_ID_Ack <> DropOff_Fix104)
				THEN
				Fix104.Discrete_In.ModelData:= Fix104_ProductData_Pers[0].Product_Model_ID;
			END_IF;
 			Fix104.NodeLayout:= Main.ECAT_Master.FixNodeLayout[104];				(*Pass in Assembled Node layout for UI*)
			Fix104.Discrete_In.Input_Node_Count:= 2;								(*Overridden for now, later version will map from UI read config sheet*)
			Fix104.Discrete_In.VB_Node_Count:= 0;								(*Overridden for now, later version will map from UI read config sheet*)
			Fix104.Discrete_In.Output_Node_Count:= 0;								(*Overridden for now, later version will map from UI read config sheet*)
			Fix104.Discrete_In.Water_Stand_Count:= 0;								(*Overridden for now, later version will map from UI read config sheet*)
			Fix104.Dry_Cycle:= GTAC_CONFIG.Dry_Cycle_Enabled;
			Fix104.Cell_In_Services:= Cell_Services_Prog.Service_Call_ForAllRobots OR In_From_ICxx.Cycle_Hold;
			Fix104.Flash_Rate:= Pulse_1S;
			(*Call FUNCTION*)
			Fix104();
			(*Output Data*)
			Out_To_ICxx.Fix104_Discrete_Image:= Fix104.Discrete_Image;


			(*Fixture 105*)
			(*Input Data*)
			Fix105.Enable_Motion:= Main.Control_Power_ON;								(*ENSURE to bind proper Relay Bank*)
			Fix105.Discrete_In:= In_From_ICxx.Fix105_Discrete_In;
			IF ((EOAT04.Part1_In_EOAT AND NOT Fix105.Load_Complete) OR Fix105.Repo_REQS.0) AND Fix105.Part_InEOAT04_1_ReadyforThisFix
				THEN
				Fix105.Discrete_In.ModelData:= EOAT04_1_ProductData_Pers.Product_Model_ID;
			ELSIF ((EOAT04.Part2_In_EOAT AND NOT Fix105.Load_Complete) OR Fix105.Repo_REQS.0) AND Fix105.Part_InEOAT04_2_ReadyforThisFix
				THEN
				Fix105.Discrete_In.ModelData:= EOAT04_2_ProductData_Pers.Product_Model_ID;
			ELSIF (Fix105.Load_Complete OR Fix105.Repo_REQS.1) AND (MAIN.R4.Task_ID_Ack <> DropOff_Fix105)
				THEN
				Fix105.Discrete_In.ModelData:= Fix105_ProductData_Pers.Product_Model_ID;
			END_IF;
			Fix105.NodeLayout:= Main.ECAT_Master.FixNodeLayout[105];				(*Pass in Assembled Node layout for UI*)
			Fix105.Discrete_In.Input_Node_Count:= 2;								(*Overridden for now, later version will map from UI read config sheet*)
			Fix105.Discrete_In.VB_Node_Count:= 0;								(*Overridden for now, later version will map from UI read config sheet*)
			Fix105.Discrete_In.Output_Node_Count:= 0;								(*Overridden for now, later version will map from UI read config sheet*)
			Fix105.Discrete_In.Water_Stand_Count:= 0;								(*Overridden for now, later version will map from UI read config sheet*)
			Fix105.Dry_Cycle:= GTAC_CONFIG.Dry_Cycle_Enabled;
			Fix105.Cell_In_Services:= Cell_Services_Prog.Service_Call_ForAllRobots OR In_From_ICxx.Cycle_Hold;
			Fix105.Flash_Rate:= Pulse_1S;
			(*Call FUNCTION*)
			Fix105();
			(*Output Data*)
			Out_To_ICxx.Fix105_Discrete_Image:= Fix105.Discrete_Image;
END_ACTION

ACTION Product_Tracking:
(*Custom Product Trackng code for this machine (Bumpers Main 2403701), primarily used to transfer model and task status*)




(*------------- Transfer Data from Fix01 or 02 to EOAT04 Upon Pickup ----------------*)
(*Fix01 / 02 are 1st Geo Set fixtures on TT01*)
	(*Picked up with EOAT Side 1*)
	RPulse[1].CLK:= Fix01.Unload_Complete1_Ack;
	RPulse[1]();
	IF RPulse[1].Q
		THEN
			EOAT04_1_ProductData_Pers:= Fix01_ProductData_Pers;
			Fix01_ProductData_Pers:= Blank_ProductData_Pers;
	END_IF;

	(*Picked up with EOAT Side 1*)
	RPulse[3].CLK:= Fix02.Unload_Complete1_Ack;
	RPulse[3]();
	IF RPulse[3].Q
		THEN
			EOAT04_1_ProductData_Pers:= Fix02_ProductData_Pers;
			Fix02_ProductData_Pers:= Blank_ProductData_Pers;
	END_IF;
(*--------------------------------------------------------------------------------*)



	
	
(*------------- Transfer Data from EOAT04 to Fix101 Upon Dropoff ----------------*)
(*Fix101 is 1st Finishing Fixture*) 
	(*Placed with EOAT Side 1*)
	RPulse[5].CLK:= Fix101.Load_Complete1_Ack;
	RPulse[5]();
	IF RPulse[5].Q
		THEN
			Fix101_ProductData_Pers:= EOAT04_1_ProductData_Pers;
			EOAT04_1_ProductData_Pers:= Blank_ProductData_Pers;
	END_IF;
	(*Placed with EOAT Side 2*)
	RPulse[6].CLK:= Fix101.Load_Complete2_Ack;
	RPulse[6]();
	IF RPulse[6].Q
		THEN
			Fix101_ProductData_Pers:= EOAT04_2_ProductData_Pers;
			EOAT04_2_ProductData_Pers:= Blank_ProductData_Pers;
	END_IF;
(*------------- Transfer Data from Fix101 to EOAT04 Upon Pickup ----------------*)
	(*Picked up with EOAT Side 2*)
	RPulse[8].CLK:= Fix101.Unload_Complete1_Ack;
	RPulse[8]();
	IF RPulse[8].Q
		THEN
			EOAT04_2_ProductData_Pers:= Fix101_ProductData_Pers;
			Fix101_ProductData_Pers:= Blank_ProductData_Pers;
	END_IF;
	
	(*Blank Data in Fix101 if required by UI*)
	IF (In_From_ICxx.CustomApplication_REQS.17 AND Fix101.Tool_At_Home AND Fix101.All_Sensors_Off AND Fix101.In_Manual) 
		OR Fix101.Reset_All_Completes
		THEN
			Fix101_ProductData_Pers:= Blank_ProductData_Pers;
	END_IF;

(*--------------------------------------------------------------------------------*)


	
	
	
(*------------- Transfer Data from EOAT04 to Fix03 or Fix04 Upon Dropff ----------------*)
(*Fix03 / 04 are 2nd Geo Set + Finishing fixtures on TT02*)
	(*Placed with EOAT Side 2*)
	RPulse[10].CLK:= Fix03.Load_Robots_Complete1;
	RPulse[10]();
	IF RPulse[10].Q
		THEN
			Fix03_ProductData_Pers:= EOAT04_2_ProductData_Pers;
			EOAT04_2_ProductData_Pers:= Blank_ProductData_Pers;
	END_IF;

	(*Placed with EOAT Side 2*)
	RPulse[12].CLK:= Fix04.Load_Complete1_Ack;
	RPulse[12]();
	IF RPulse[12].Q
		THEN
			Fix04_ProductData_Pers:= EOAT04_2_ProductData_Pers;
			EOAT04_2_ProductData_Pers:= Blank_ProductData_Pers;
	END_IF;

	(*Blank Data in EOAT04 Side 1*)
	IF In_From_ICxx.CustomApplication_REQS.29 AND MAIN.R4.At_Home AND EOAT04.EOAT_Part1_Empty
		THEN
			EOAT04_1_ProductData_Pers:= Blank_ProductData_Pers;
	END_IF;

	(*Blank Data in EOAT04 Side 2*)
	IF In_From_ICxx.CustomApplication_REQS.30 AND MAIN.R4.At_Home AND EOAT04.EOAT_Part2_Empty
		THEN
			EOAT04_2_ProductData_Pers:= Blank_ProductData_Pers;
	END_IF;

	(*Blank EOAT04 Data in event of a full empty check*)
	RPulse[13].CLK:= EOAT04.CMD_CheckAllSensors_OFF AND EOAT04.EOAT_Part1_Empty AND EOAT04.EOAT_Part2_Empty;
	RPulse[13]();
	IF RPulse[13].Q
		THEN
			EOAT04_1_ProductData_Pers:= Blank_ProductData_Pers;
			EOAT04_2_ProductData_Pers:= Blank_ProductData_Pers;
	END_IF;
	
(*--------------------------------------------------------------------------------*)


(*------------- Transfer Data from Fix03 or 04 to EOAT04 Pickup ----------------*)
	(*Picked up with EOAT Side 1*)
	RPulse[14].CLK:= Fix03.Unload_Complete1_Ack;
	RPulse[14]();
	IF RPulse[14].Q
		THEN
			EOAT04_1_ProductData_Pers:= Fix03_ProductData_Pers;
			Fix03_ProductData_Pers:= Blank_ProductData_Pers;
	END_IF;

	(*Picked up with EOAT Side 1*)
	RPulse[16].CLK:= Fix04.Unload_Complete1_Ack;
	RPulse[16]();
	IF RPulse[16].Q
		THEN
			EOAT04_1_ProductData_Pers:= Fix04_ProductData_Pers;
			Fix04_ProductData_Pers:= Blank_ProductData_Pers;
	END_IF;
	
   (*Blank Data in Fix03*)
	IF (In_From_ICxx.CustomApplication_REQS.3 AND Fix03.Tool_At_Home AND Fix03.All_Sensors_Off AND Fix03.In_Manual) 
		THEN
			Fix03_ProductData_Pers:= Blank_ProductData_Pers;
	END_IF;

	(*Blank Data in Fix04*)
	IF (In_From_ICxx.CustomApplication_REQS.4 AND Fix04.Tool_At_Home AND Fix04.All_Sensors_Off AND Fix04.In_Manual) 
		THEN
			Fix04_ProductData_Pers:= Blank_ProductData_Pers;
	END_IF;

(*--------------------------------------------------------------------------------*)
	
	
	
	
	
(*------------- Transfer Data from EOAT04 to Fix102 Upon Dropoff ----------------*)
(*Fix102 is Insepction Area*)
	(*Placed with EOAT Side 1*)
	RPulse[18].CLK:= Fix102.Load_Complete1_Ack;
	RPulse[18]();
	IF RPulse[18].Q
		THEN
			Fix102_ProductData_Pers:= EOAT04_1_ProductData_Pers;
			EOAT04_1_ProductData_Pers:= Blank_ProductData_Pers;
	END_IF;
	
(*------------- Transfer Data from FIX102 to EOAT04 Upon Pickup ----------------*)
	(*Picked up with EOAT Side 2*)
	RPulse[20].CLK:= Fix102.Unload_Complete1_Ack;
	RPulse[20]();
	IF RPulse[20].Q
		THEN
			EOAT04_2_ProductData_Pers:= Fix102_ProductData_Pers;
			Fix102_ProductData_Pers:= Blank_ProductData_Pers;
	END_IF;
	(*Picked up with EOAT Side 1*)
	RPulse[21].CLK:= Fix102.Unload_Complete2_Ack;
	RPulse[21]();
	IF RPulse[21].Q
		THEN
			EOAT04_1_ProductData_Pers:= Fix102_ProductData_Pers;
			Fix102_ProductData_Pers:= Blank_ProductData_Pers;
	END_IF;
		
	(*Blank Data in Fix102*)
	IF (In_From_ICxx.CustomApplication_REQS.18 AND Fix102.Tool_At_Home AND Fix102.All_Sensors_Off AND Fix102.In_Manual) 
		OR Fix102.Reset_All_Completes
			THEN
			Fix102_ProductData_Pers:= Blank_ProductData_Pers;
	END_IF;

(*--------------------------------------------------------------------------------*)

	
	
	
	
(*------------- Transfer Data from Fix05 to EOAT04 Upon Pickup ----------------*)
(*Fix05 is Rework Insert only station*)
	(*Picked up with EOAT Side 1*)
	RPulse[22].CLK:= Fix05.Unload_Complete1_Ack;
	RPulse[22]();
	IF RPulse[22].Q
		THEN
			EOAT04_1_ProductData_Pers:= Fix05_ProductData_Pers;
			Fix05_ProductData_Pers:= Blank_ProductData_Pers;
	END_IF;
	(*Picked up with EOAT Side 2*)
	RPulse[23].CLK:= Fix05.Unload_Complete2_Ack;
	RPulse[23]();
	IF RPulse[23].Q
		THEN
			EOAT04_2_ProductData_Pers:= Fix05_ProductData_Pers;
			Fix05_ProductData_Pers:= Blank_ProductData_Pers;
	END_IF;
(*--------------------------------------------------------------------------------*)
	
	
	

(*------------- Transfer Data from EOAT04 to Fix103 Upon Dropoff ----------------*)
(*Fix103 is QA Request / NOK Offload only station*)
	(*Placed with EOAT Side 1*)
	RPulse[24].CLK:= Fix103.Load_Complete1_Ack;
	RPulse[24]();
	IF RPulse[24].Q
		THEN
			Fix103_ProductData_Pers:= EOAT04_2_ProductData_Pers;
			EOAT04_2_ProductData_Pers:= Blank_ProductData_Pers;
	END_IF;
	(*Placed with EOAT Side 2*)
	RPulse[25].CLK:= Fix103.Load_Complete2_Ack;
	RPulse[25]();
	IF RPulse[25].Q
		THEN
			Fix103_ProductData_Pers:= EOAT04_2_ProductData_Pers;
			EOAT04_1_ProductData_Pers:= Blank_ProductData_Pers;
	END_IF;
	
	(*Blank Data in Fix103*)
	IF (In_From_ICxx.CustomApplication_REQS.19 AND Fix103.Tool_At_Home AND Fix103.All_Sensors_Off AND Fix103.In_Manual) 
		OR Fix103.Reset_All_Completes
			THEN
			Fix103_ProductData_Pers:= Blank_ProductData_Pers;
	END_IF;

(*--------------------------------------------------------------------------------*)

	
	
	
(*------------- Transfer Data from EOAT04 to Fix104 Upon Dropoff ----------------*)
(*Fix104 is Buffer to load finished parts on if Paint is down*)
	(*Placed with EOAT Side 1*)
	RPulse[26].CLK:= Fix104.Load_Complete1_Ack;
	RPulse[26]();
	IF RPulse[26].Q
		THEN
			IF (Fix104.Fix_ID >=1 AND  Fix104.Fix_ID<=5)
				THEN
					Fix104_ProductData_Pers[Fix104.Fix_ID]:= EOAT04_1_ProductData_Pers;
					EOAT04_1_ProductData_Pers:= Blank_ProductData_Pers;
				END_IF
	END_IF;	
	(*Placed with EOAT Side 2*)
	RPulse[27].CLK:= Fix104.Load_Complete2_Ack;
	RPulse[27]();
	IF RPulse[27].Q
		THEN
			IF (Fix104.Fix_ID >=1 AND  Fix104.Fix_ID<=5)
				THEN
					Fix104_ProductData_Pers[Fix104.Fix_ID]:= EOAT04_2_ProductData_Pers;
					EOAT04_2_ProductData_Pers:= Blank_ProductData_Pers;
				END_IF
	END_IF;	
	
	(*Blank Data in Fix104*)
	IF (In_From_ICxx.CustomApplication_REQS.20 AND Fix104.Tool_At_Home AND Fix104.All_Sensors_Off AND Fix104.In_Manual) 
		OR Fix104.Reset_All_Completes
			THEN
			Fix104_ProductData_Pers[0]:= Blank_ProductData_Pers;
	END_IF;

(*--------------------------------------------------------------------------------*)




	
(*------------- Transfer Data from EOAT04 to Fix105 Upon Dropoff ----------------*)
(*Fix105 is final offload to Paint*)
	(*Placed with EOAT Side 1*)
	RPulse[28].CLK:= Fix105.Load_Complete1_Ack;
	RPulse[28]();
	IF RPulse[28].Q
		THEN
			Fix105_ProductData_Pers:= EOAT04_1_ProductData_Pers;
			EOAT04_1_ProductData_Pers:= Blank_ProductData_Pers;
	END_IF;	
	(*Placed with EOAT Side 2*)
	RPulse[29].CLK:= Fix105.Load_Complete2_Ack;
	RPulse[29]();
	IF RPulse[29].Q
		THEN
			Fix105_ProductData_Pers:= EOAT04_2_ProductData_Pers;
			EOAT04_2_ProductData_Pers:= Blank_ProductData_Pers;
	END_IF;	
	
	(*Blank Data in Fix105*)
	IF (In_From_ICxx.CustomApplication_REQS.21 AND Fix105.Tool_At_Home AND Fix105.All_Sensors_Off AND Fix105.In_Manual) 
		OR Fix105.Reset_All_Completes
			THEN
			Fix105_ProductData_Pers:= Blank_ProductData_Pers;
	END_IF;

(*--------------------------------------------------------------------------------*)
END_ACTION

ACTION Robots:



(*R1 ------------------------*)
		(*Input Data*)
		R1.FB_In.Robot_Type:=KUKA_KRC4_SAFEOP_TurnTable;
		R1.FB_In.Install_Zero_Orientation:= 180; 	(*Set this value between 0 and 359 to set the zero position of the robot physical install with reference to 12 o'clock symbol on UI screens*)
		R1.FB_In.Under_Construction:= GTAC_CONFIG.Under_Construction;
		R1.FB_In.In_SIM_Mode:= GTAC_CONFIG.In_SIM_Mode;
		R1.FB_In.SIM_StartWorkAround:= FALSE;  (*Main.SIM_WorkAround_StartRobots*)
		R1.FB_In.CoE_Read_Trigger:= (GTAC_CONFIG.Option_Robot_Count>=1) AND Pulse_CoERead;
		R1.FB_In.Ecat_Master_AmsNetID:= MAIN.ECAT_Master.AmsID;
		R1.FB_In.Prev_EcatNode_Present:= NOT MD01.EP1918_NotPresent; (*Ensure Previous Node Exists to determine Ecat Cable Break of this Devices Input Cable*)
		R1.FB_In.Safety_RST:=SAFETY_RESET;
		R1.FB_In.Enable_Motion:= All_Estops_OK OR GTAC_CONFIG.Under_Construction;
		R1.FB_In.Alarm_RST:=In_From_ICxx.ControlPower1;
		R1.FB_In.Select_Play:=FALSE;
		R1.FB_In.Select_Teach:=FALSE;
		R1.FB_In.Select_Remote:=FALSE;
		R1.FB_In.Start_Scan:=In_From_ICxx.StartRobots;
		R1.FB_In.Stop_Scan:=In_From_ICxx.StopRobots;
		R1.FB_In.Stop_Scan2:=FALSE;
		R1.FB_In.In_DryCycle:= GTAC_CONFIG.Dry_Cycle_Enabled;
		R1.FB_In.Low_Speed:= GTAC_CONFIG.Low_Speed_Enabled;
		R1.FB_In.Speed_Request:= In_From_ICxx.Global_Robot_Speed;
		R1.FB_In.Force_MasterTest_Req:= Cell_Services_Prog.Human_Reqs_MasterTest OR Cell_Services_Prog.A_Robot_Reqs_MasterTest;
		R1.FB_In.Force_BrakeTest_Req:= Cell_Services_Prog.Human_Reqs_BrakeTest OR Cell_Services_Prog.A_Robot_Reqs_BrakeTest;
		R1.FB_In.Major_Faults:= Faults.System_Major_Fault;
		R1.FB_In.Teach_Interlock:=R1_Data.Teach_Interlock;
		R1.FB_In.Weld_Inhibit:=In_From_ICxx.Rxx_Weld_Inhibit;
		R1.FB_In.Option_Disable_WaterFLT:= FALSE AND GTAC_CONFIG.Under_Construction OR (MAIN.R1.Task_ID_Ack=Tip_Change_EXT); (*Used to disable water fault if no water is present. use with caution*)
		R1.FB_In.OK_ToEnter_EquipInterf1:=R1_Data.OK_ToEnter_EquipInterf1;
		R1.FB_In.OK_ToEnter_EquipInterf2:=R1_Data.OK_ToEnter_EquipInterf2;
		R1.FB_In.OK_ToEnter_EquipInterf3:=R1_Data.OK_ToEnter_EquipInterf3;
		R1.FB_In.OK_ToEnter_EquipInterf4:=R1_Data.OK_ToEnter_EquipInterf4;
		R1.FB_In.OK_ToEnter_EquipInterf5:=R1_Data.OK_ToEnter_EquipInterf5;
		R1.FB_In.OK_ToEnter_EquipInterf6:=R1_Data.OK_ToEnter_EquipInterf6;
		R1.FB_In.OK_ToEnter_EquipInterf7:=R1_Data.OK_ToEnter_EquipInterf7;
		R1.FB_In.OK_ToEnter_EquipInterf8:=R1_Data.OK_ToEnter_EquipInterf8;
		R1.FB_In.OK_ToEnter_EquipInterf9:=R1_Data.OK_ToEnter_EquipInterf9;
		R1.FB_In.OK_ToEnter_HumanInterf1:=R1_Data.OK_ToEnter_HumanInterf1;
		R1.FB_In.OK_ToEnter_HumanInterf2:=R1_Data.OK_ToEnter_HumanInterf2;
		R1.FB_In.OK_ToEnter_HumanInterf3:=R1_Data.OK_ToEnter_HumanInterf3;
		R1.FB_In.OK_ToEnter_HumanInterf4:=R1_Data.OK_ToEnter_HumanInterf4;
		R1.FB_In.OK_ToEnter_HumanInterf5:=R1_Data.OK_ToEnter_HumanInterf5;
		R1.FB_In.OK_ToEnter_HumanInterf6:=R1_Data.OK_ToEnter_HumanInterf6;
		R1.FB_In.OK_ToEnter_HumanInterf7:=R1_Data.OK_ToEnter_HumanInterf7;
		R1.FB_In.OK_ToEnter_HumanInterf8:=R1_Data.OK_ToEnter_HumanInterf8;
		R1.FB_In.OK_ToEnter_RobotInterfs:= R1_Data.OK_ToEnter_RobotInterfs;
		R1.FB_In.Fix_ID:= R1_Data.Fix_ID[R1.Location_Index];
		R1.FB_In.Model_ID:= R1_Data.Model_ID[R1.Location_Index];
		R1.FB_In.Task_ID:= R1_Data.Task_ID[R1.Location_Index];
		R1.FB_In.Proceed_From_Pounce:= R1_Data.Proceed_From_Pounce[R1.Location_Index];
		R1.FB_In.Complete_Ack:= R1_Data.Complete_Ack[R1.Location_Index];
		R1.FB_In.PeripheralReq_Ack:= R1_Data.PeripheralReq_Ack[R1.Location_Index];
		R1.FB_In.AuxReq_Ack:= R1_Data.AuxReq_Ack[R1.Location_Index];
		R1.FB_In.User_Inputs.0:= R2.User_Outputs.0 AND R3.User_Outputs.0; (*confirm table position to weld main*)
		R1.FB_In.User_Inputs.1:= NOT R2.User_Outputs.1 AND R3.User_Outputs.1; (*confirm table position to weld subs*)
		R1.FB_In.User_Inputs.2:= R2.User_Outputs.2 AND R3.User_Outputs.2;
		R1.FB_In.User_Inputs.3:= R2.User_Outputs.2 AND R3.User_Outputs.2 AND R2.User_Outputs.3;
		R1.FB_In.User_Inputs.4:= FALSE;
		R1.FB_In.User_Inputs.5:= FALSE;
		R1.FB_In.User_Inputs.6:= FALSE;
		R1.FB_In.User_Inputs.7:= FALSE;
			(*Configure Options Amounts*)
			R1.FB_In.Options.WeldCont_Amount:=0; 					(*Select amount of Spot Type Weld Controllers here (0 min, 4 max)*)
			R1.FB_In.Options.WaterStand_Amount:= 0;				(*Select amount of Water Stands here (0 min, 2 max)*)
			R1.FB_In.Options.MIGCont_Amount:= 1;					(*Select amount of MIG Type Weld Controllers here (0 min, 1 max)*)
			R1.FB_In.Options.Reamer_Amount:= 1;					(*Select amount of Tip Reamers here (0 min, 1 max)*)
			R1.FB_In.Options.EOAT_Amount:= 0;						(*Assign EOAT number to robot (0 min, 10 max)*)
			(*Configure Options Parameters*)
			
			(*R1.Reamer[1](
				(*FB Inputs*)
					Enable_Motion:= All_Estops_OK,
					Fronius_Ream:= TRUE,
                    Binzel_Ream:= FALSE,  (*optional*)
					Ream_REQ:= R1.Peripheral_Req.5 AND (R1.Task_ID_Ack=Tip_Dress),

				(*FB Outputs*)
					Reaming_Complete=> ,(*mapped in cell services*)
					);*)
					
			R1.Reamer[1](
				(*FB Inputs*)
					Enable_Motion:= All_Estops_OK,
					Fronius_Ream:= TRUE,
                    Binzel_Ream:= FALSE,  (*optional*)
					
					Ream_REQ:= R1.Peripheral_Req.1 AND ((R1.Task_ID_Ack=Tip_Dress)OR (R1.In_T1 AND R1.Peripheral_Req.5)),
					Ream_Time:= T#2S,
					Ream_Clamp_Open:= R1.Reamer[1].N01.I.1,
					Spray_REQ:= R1.Peripheral_Req.2 AND ((R1.Task_ID_Ack=Tip_Dress)OR (R1.In_T1 AND R1.Peripheral_Req.5)),
					Spray_Time:= T#2S,
					F_WireCutter_REQ:= R1.Peripheral_Req.4 AND ((R1.Task_ID_Ack=Tip_Dress)OR (R1.In_T1 AND R1.Peripheral_Req.5)),
					F_WireCutter_Time:= T#1S,
					
				(*FB Outputs*)
					Reaming_Complete=> ,(*mapped in cell services*)
					(*The following are for Binzel type reamers only*)
					LifterUp_ACK=> , (*mapped in cell services*)
					Clamp_ACK=>,(*mapped in cell services*)
					Injector_ACK=> ,(*mapped in cell services*)
					WireCutter_ACK=> (*mapped in cell services*)
					);		
		(*Call Actual Object*)
		R1();
		(*Output Data*)
		Out_To_ICxx.Robot[1].Robot_Type:= R1.FB_In.Robot_Type;
		Out_To_ICxx.Robot[1].Status:= R1.Status;
		Out_To_ICxx.Robot[1].Axis_Data[1]:= R1.S_Axis_Pos_Raw; 
		Out_To_ICxx.Robot[1].In_Image:= R1.Input_Image;
		Out_To_ICxx.Robot[1].Out_Image:= R1.Output_Image;
		Out_To_ICxx.Robot[1].Discrete_ImageFSOE:= R1.Discrete_Image_FSoE;
		Out_To_ICxx.Robot[1].Options:= R1.FB_In.Options;
			Out_To_ICxx.Robot[1].WS_Discrete_Image[1]:= R1.WS[1].Discrete_Image;
			Out_To_ICxx.Robot[1].WS_Discrete_Image[2]:= R1.WS[2].Discrete_Image;
 			Out_To_ICxx.Robot[1].ATI_Discrete_Image:= R1.ATI[1].Discrete_Image;
			Out_To_ICxx.Robot[1].Reamer_Discrete_Image:= R1.Reamer[1].Discrete_Image;
			Out_To_ICxx.Robot[1].Fronius_Status:= R1.Fronius_Status;
		Out_To_ICxx.Robot[1].Ped_IO_ToShow[1]:= 0;			(*Set to Ped value if this robots ecat string contains the Ped's IO*)
		Out_To_ICxx.Robot[1].Ped_IO_ToShow[2]:= 0;			(*Set to Ped value if this robots ecat string contains the Ped's IO*)
		Out_To_ICxx.Robot[1].ECAT_Cable_Breaks:= R1.ECatSlave_Cable_Breaks;
		Out_To_ICxx.Robot[1].CT:= R1.CT;
		(*Example of passing Turntable Axis Data*)
		//Out_To_ICxx.TT01_Location_Index:= R1.TT_Axis_Location_Index; (*Pass Turntable location*) DEBUG - RESTORE AFTER SIM - RJ
		
		(*IF (MAIN.SIM_WorkAround_TT01_Position_Index[0] = TRUE)
			THEN Out_To_ICxx.TT01_Location_Index:= 1;
		ELSIF (MAIN.SIM_WorkAround_TT01_Position_Index[1] = TRUE)
			THEN Out_To_ICxx.TT01_Location_Index:= 2;
		ELSE
			Out_To_ICxx.TT01_Location_Index:= 0;
		END_IF*)	//DEBUG - RJ - REMOVE ABOVE AFTER SIM, RESTORE original
		Out_To_ICxx.TT01_Location_Index:= R1.TT_Axis_Location_Index;


(*R2 ------------------------*)
		(*Input Data*)
		R2.FB_In.Robot_Type:=KUKA_KRC4_SAFEOP;
		R2.FB_In.Install_Zero_Orientation:= 180; 	(*Set this value between 0 and 359 to set the zero position of the robot physical install with reference to 12 o'clock symbol on UI screens*)
		R2.FB_In.Under_Construction:= GTAC_CONFIG.Under_Construction;
		R2.FB_In.In_SIM_Mode:= GTAC_CONFIG.In_SIM_Mode;
		R2.FB_In.SIM_StartWorkAround:= FALSE;  (*Main.SIM_WorkAround_StartRobots*)
		R2.FB_In.CoE_Read_Trigger:= (GTAC_CONFIG.Option_Robot_Count>=2) AND Pulse_CoERead;
		R2.FB_In.Ecat_Master_AmsNetID:= MAIN.ECAT_Master.AmsID;
		R2.FB_In.Prev_EcatNode_Present:= NOT R1.EK1100_NotPresent; (*Ensure Previous Node Exists to determine Ecat Cable Break of this Devices Input Cable*)
		R2.FB_In.Safety_RST:=SAFETY_RESET;
		R2.FB_In.Enable_Motion:= All_Estops_OK OR GTAC_CONFIG.Under_Construction;
		R2.FB_In.Alarm_RST:=In_From_ICxx.ControlPower1;
		R2.FB_In.Select_Play:=FALSE;
		R2.FB_In.Select_Teach:=FALSE;
		R2.FB_In.Select_Remote:=FALSE;
		R2.FB_In.Start_Scan:=In_From_ICxx.StartRobots;
		R2.FB_In.Stop_Scan:=In_From_ICxx.StopRobots;
		R2.FB_In.Stop_Scan2:=FALSE;
		R2.FB_In.In_DryCycle:= GTAC_CONFIG.Dry_Cycle_Enabled;
		R2.FB_In.Low_Speed:= GTAC_CONFIG.Low_Speed_Enabled;
		R2.FB_In.Speed_Request:= In_From_ICxx.Global_Robot_Speed;
		R2.FB_In.Force_MasterTest_Req:= Cell_Services_Prog.Human_Reqs_MasterTest OR Cell_Services_Prog.A_Robot_Reqs_MasterTest;
		R2.FB_In.Force_BrakeTest_Req:= Cell_Services_Prog.Human_Reqs_BrakeTest OR Cell_Services_Prog.A_Robot_Reqs_BrakeTest;
		R2.FB_In.Major_Faults:= Faults.System_Major_Fault;
		R2.FB_In.Teach_Interlock:=R2_Data.Teach_Interlock;
		R2.FB_In.Weld_Inhibit:=In_From_ICxx.Rxx_Weld_Inhibit;
		R2.FB_In.Option_Disable_WaterFLT:= FALSE AND GTAC_CONFIG.Under_Construction OR (MAIN.R2.Task_ID_Ack=Tip_Change_EXT); (*Used to disable water fault if no water is present. use with caution*)
		R2.FB_In.OK_ToEnter_EquipInterf1:=R2_Data.OK_ToEnter_EquipInterf1;
		R2.FB_In.OK_ToEnter_EquipInterf2:=R2_Data.OK_ToEnter_EquipInterf2;
		R2.FB_In.OK_ToEnter_EquipInterf3:=R2_Data.OK_ToEnter_EquipInterf3;
		R2.FB_In.OK_ToEnter_EquipInterf4:=R2_Data.OK_ToEnter_EquipInterf4;
		R2.FB_In.OK_ToEnter_EquipInterf5:=R2_Data.OK_ToEnter_EquipInterf5;
		R2.FB_In.OK_ToEnter_EquipInterf6:=R2_Data.OK_ToEnter_EquipInterf6;
		R2.FB_In.OK_ToEnter_EquipInterf7:=R2_Data.OK_ToEnter_EquipInterf7;
		R2.FB_In.OK_ToEnter_EquipInterf8:=R2_Data.OK_ToEnter_EquipInterf8;
		R2.FB_In.OK_ToEnter_EquipInterf9:=R2_Data.OK_ToEnter_EquipInterf9;
		R2.FB_In.OK_ToEnter_HumanInterf1:=R2_Data.OK_ToEnter_HumanInterf1;
		R2.FB_In.OK_ToEnter_HumanInterf2:=R2_Data.OK_ToEnter_HumanInterf2;
		R2.FB_In.OK_ToEnter_HumanInterf3:=R2_Data.OK_ToEnter_HumanInterf3;
		R2.FB_In.OK_ToEnter_HumanInterf4:=R2_Data.OK_ToEnter_HumanInterf4;
		R2.FB_In.OK_ToEnter_HumanInterf5:=R2_Data.OK_ToEnter_HumanInterf5;
		R2.FB_In.OK_ToEnter_HumanInterf6:=R2_Data.OK_ToEnter_HumanInterf6;
		R2.FB_In.OK_ToEnter_HumanInterf7:=R2_Data.OK_ToEnter_HumanInterf7;
		R2.FB_In.OK_ToEnter_HumanInterf8:=R2_Data.OK_ToEnter_HumanInterf8;
		R2.FB_In.OK_ToEnter_RobotInterfs:= R2_Data.OK_ToEnter_RobotInterfs;
		R2.FB_In.Fix_ID:=R2_Data.Fix_ID[R2.Location_Index];
		R2.FB_In.Model_ID:=R2_Data.Model_ID[R2.Location_Index];
		R2.FB_In.Task_ID:=R2_Data.Task_ID[R2.Location_Index];
		R2.FB_In.Proceed_From_Pounce:=R2_Data.Proceed_From_Pounce[R2.Location_Index];
		R2.FB_In.Complete_Ack:=R2_Data.Complete_Ack[R2.Location_Index];
		R2.FB_In.PeripheralReq_Ack:=R2_Data.PeripheralReq_Ack[R2.Location_Index];
		R2.FB_In.AuxReq_Ack:= R2_Data.AuxReq_Ack[R2.Location_Index];
		R2.FB_In.User_Inputs.0:= R1.User_Outputs.0;
		R2.FB_In.User_Inputs.1:= FALSE;
		R2.FB_In.User_Inputs.2:= R1.User_Outputs.2;
		R2.FB_In.User_Inputs.3:= R1.User_Outputs.3;
		R2.FB_In.User_Inputs.4:= FALSE;
		R2.FB_In.User_Inputs.5:= FALSE;
		R2.FB_In.User_Inputs.6:= FALSE;
		R2.FB_In.User_Inputs.7:= FALSE;
			(*Configure Options Amounts*)
			R2.FB_In.Options.WeldCont_Amount:=0; 					(*Select amount of Spot Type Weld Controllers here (0 min, 4 max)*)
			R2.FB_In.Options.WaterStand_Amount:= 0;				(*Select amount of Water Stands here (0 min, 2 max)*)
			R2.FB_In.Options.MIGCont_Amount:= 1;					(*Select amount of MIG Type Weld Controllers here (0 min, 1 max)*)
			R2.FB_In.Options.Reamer_Amount:= 1;					(*Select amount of Tip Reamers here (0 min, 1 max)*)
			R2.FB_In.Options.EOAT_Amount:= 0;						(*Assign EOAT number to robot (0 min, 10 max)*)
			(*Configure Options Parameters*)

			R2.Reamer[1](
				(*FB Inputs*)
					Enable_Motion:= All_Estops_OK,
					Fronius_Ream:= TRUE,
                    Binzel_Ream:= FALSE,  (*optional*)
					
					Ream_REQ:= R2.Peripheral_Req.1 AND ((R2.Task_ID_Ack=Tip_Dress)OR (R2.In_T1 AND R2.Peripheral_Req.5)),
					Ream_Time:= T#2S,
					Ream_Clamp_Open:= R2.Reamer[1].N01.I.1,
					Spray_REQ:= R2.Peripheral_Req.2 AND ((R2.Task_ID_Ack=Tip_Dress)OR (R2.In_T1 AND R2.Peripheral_Req.5)),
					Spray_Time:= T#2S,
					F_WireCutter_REQ:= R2.Peripheral_Req.4 AND ((R2.Task_ID_Ack=Tip_Dress)OR (R2.In_T1 AND R2.Peripheral_Req.5)),
					F_WireCutter_Time:= T#1S,
					
				(*FB Outputs*)
					Reaming_Complete=> ,(*mapped in cell services*)
					(*The following are for Binzel type reamers only*)
					LifterUp_ACK=> , (*mapped in cell services*)
					Clamp_ACK=>,(*mapped in cell services*)
					Injector_ACK=> ,(*mapped in cell services*)
					WireCutter_ACK=> (*mapped in cell services*)
					);
			
			(*R2.Reamer[1](
				(*FB Inputs*)
					Enable_Motion:= All_Estops_OK,
					Fronius_Ream:= TRUE,
                    Binzel_Ream:= FALSE,  (*optional*)
					Ream_REQ:= R2.Peripheral_Req.5 AND (R2.Task_ID_Ack=Tip_Dress),

				(*FB Outputs*)
					Reaming_Complete=> ,(*mapped in cell services*)
					);*)
		(*Call Actual Object*)
		R2();
		(*Output Data*)
		Out_To_ICxx.Robot[2].Robot_Type:= R2.FB_In.Robot_Type;
		Out_To_ICxx.Robot[2].Status:= R2.Status;
		Out_To_ICxx.Robot[2].Axis_Data[1]:= R2.S_Axis_Pos_Raw;
		Out_To_ICxx.Robot[2].In_Image:= R2.Input_Image;
		Out_To_ICxx.Robot[2].Out_Image:= R2.Output_Image;
		Out_To_ICxx.Robot[2].Discrete_ImageFSOE:= R2.Discrete_Image_FSoE;
		Out_To_ICxx.Robot[2].Options:= R2.FB_In.Options;
			Out_To_ICxx.Robot[2].WS_Discrete_Image[1]:= R2.WS[1].Discrete_Image;
			Out_To_ICxx.Robot[2].WS_Discrete_Image[2]:= R2.WS[2].Discrete_Image;
 			Out_To_ICxx.Robot[2].ATI_Discrete_Image:= R2.ATI[1].Discrete_Image;
			Out_To_ICxx.Robot[2].Reamer_Discrete_Image:= R2.Reamer[1].Discrete_Image;
			Out_To_ICxx.Robot[2].Fronius_Status:= R2.Fronius_Status;
		Out_To_ICxx.Robot[2].Ped_IO_ToShow[1]:= 0;			(*Set to Ped value if this robots ecat string contains the Ped's IO*)
		Out_To_ICxx.Robot[2].Ped_IO_ToShow[2]:= 0;			(*Set to Ped value if this robots ecat string contains the Ped's IO*)
		Out_To_ICxx.Robot[2].ECAT_Cable_Breaks:= R2.ECatSlave_Cable_Breaks;
		Out_To_ICxx.Robot[2].CT:= R2.CT;



(*R3 ------------------------*)
		(*Input Data*)
		R3.FB_In.Robot_Type:=KUKA_KRC4_SAFEOP;
		R3.FB_In.Install_Zero_Orientation:= 180; 	(*Set this value between 0 and 359 to set the zero position of the robot physical install with reference to 12 o'clock symbol on UI screens*)
		R3.FB_In.Under_Construction:= GTAC_CONFIG.Under_Construction;
		R3.FB_In.In_SIM_Mode:= GTAC_CONFIG.In_SIM_Mode;
		R3.FB_In.SIM_StartWorkAround:= FALSE;  (*Main.SIM_WorkAround_StartRobots*)
		R3.FB_In.CoE_Read_Trigger:= (GTAC_CONFIG.Option_Robot_Count>=3) AND Pulse_CoERead;
		R3.FB_In.Ecat_Master_AmsNetID:= MAIN.ECAT_Master.AmsID;
		R3.FB_In.Prev_EcatNode_Present:= NOT R2.EK1100_NotPresent; (*Ensure Previous Node Exists to determine Ecat Cable Break of this Devices Input Cable*)
		R3.FB_In.Safety_RST:=SAFETY_RESET;
		R3.FB_In.Enable_Motion:= All_Estops_OK OR GTAC_CONFIG.Under_Construction;
		R3.FB_In.Alarm_RST:=In_From_ICxx.ControlPower1;
		R3.FB_In.Select_Play:=FALSE;
		R3.FB_In.Select_Teach:=FALSE;
		R3.FB_In.Select_Remote:=FALSE;
		R3.FB_In.Start_Scan:=In_From_ICxx.StartRobots;
		R3.FB_In.Stop_Scan:=In_From_ICxx.StopRobots;
		R3.FB_In.Stop_Scan2:=FALSE;
		R3.FB_In.In_DryCycle:= GTAC_CONFIG.Dry_Cycle_Enabled;
		R3.FB_In.Low_Speed:= GTAC_CONFIG.Low_Speed_Enabled;
		R3.FB_In.Speed_Request:= In_From_ICxx.Global_Robot_Speed;
		R3.FB_In.Force_MasterTest_Req:= Cell_Services_Prog.Human_Reqs_MasterTest OR Cell_Services_Prog.A_Robot_Reqs_MasterTest;
		R3.FB_In.Force_BrakeTest_Req:= Cell_Services_Prog.Human_Reqs_BrakeTest OR Cell_Services_Prog.A_Robot_Reqs_BrakeTest;
		R3.FB_In.Major_Faults:= Faults.System_Major_Fault;
		R3.FB_In.Teach_Interlock:=R3_Data.Teach_Interlock;
		R3.FB_In.Weld_Inhibit:=In_From_ICxx.Rxx_Weld_Inhibit;
		R3.FB_In.Option_Disable_WaterFLT:= FALSE AND GTAC_CONFIG.Under_Construction OR (MAIN.R3.Task_ID_Ack=Tip_Change_EXT); (*Used to disable water fault if no water is present. use with caution*)
		R3.FB_In.OK_ToEnter_EquipInterf1:=R3_Data.OK_ToEnter_EquipInterf1;
		R3.FB_In.OK_ToEnter_EquipInterf2:=R3_Data.OK_ToEnter_EquipInterf2;
		R3.FB_In.OK_ToEnter_EquipInterf3:=R3_Data.OK_ToEnter_EquipInterf3;
		R3.FB_In.OK_ToEnter_EquipInterf4:=R3_Data.OK_ToEnter_EquipInterf4;
		R3.FB_In.OK_ToEnter_EquipInterf5:=R3_Data.OK_ToEnter_EquipInterf5;
		R3.FB_In.OK_ToEnter_EquipInterf6:=R3_Data.OK_ToEnter_EquipInterf6;
		R3.FB_In.OK_ToEnter_EquipInterf7:=R3_Data.OK_ToEnter_EquipInterf7;
		R3.FB_In.OK_ToEnter_EquipInterf8:=R3_Data.OK_ToEnter_EquipInterf8;
		R3.FB_In.OK_ToEnter_EquipInterf9:=R3_Data.OK_ToEnter_EquipInterf9;
		R3.FB_In.OK_ToEnter_HumanInterf1:=R3_Data.OK_ToEnter_HumanInterf1;
		R3.FB_In.OK_ToEnter_HumanInterf2:=R3_Data.OK_ToEnter_HumanInterf2;
		R3.FB_In.OK_ToEnter_HumanInterf3:=R3_Data.OK_ToEnter_HumanInterf3;
		R3.FB_In.OK_ToEnter_HumanInterf4:=R3_Data.OK_ToEnter_HumanInterf4;
		R3.FB_In.OK_ToEnter_HumanInterf5:=R3_Data.OK_ToEnter_HumanInterf5;
		R3.FB_In.OK_ToEnter_HumanInterf6:=R3_Data.OK_ToEnter_HumanInterf6;
		R3.FB_In.OK_ToEnter_HumanInterf7:=R3_Data.OK_ToEnter_HumanInterf7;
		R3.FB_In.OK_ToEnter_HumanInterf8:=R3_Data.OK_ToEnter_HumanInterf8;
		R3.FB_In.OK_ToEnter_RobotInterfs:= R3_Data.OK_ToEnter_RobotInterfs;
		R3.FB_In.Fix_ID:=R3_Data.Fix_ID[R3.Location_Index];
		R3.FB_In.Model_ID:=R3_Data.Model_ID[R3.Location_Index];
		R3.FB_In.Task_ID:=R3_Data.Task_ID[R3.Location_Index];
		R3.FB_In.Proceed_From_Pounce:=R3_Data.Proceed_From_Pounce[R3.Location_Index];
		R3.FB_In.Complete_Ack:=R3_Data.Complete_Ack[R3.Location_Index];
		R3.FB_In.PeripheralReq_Ack:=R3_Data.PeripheralReq_Ack[R3.Location_Index];
		R3.FB_In.AuxReq_Ack:=R3_Data.AuxReq_Ack[R3.Location_Index];
		R3.FB_In.User_Inputs.0:= R1.User_Outputs.0;
		R3.FB_In.User_Inputs.1:= R1.User_Outputs.1;
		R3.FB_In.User_Inputs.2:= R1.User_Outputs.2;
		R3.FB_In.User_Inputs.3:= FALSE;
		R3.FB_In.User_Inputs.4:= FALSE;
		R3.FB_In.User_Inputs.5:= FALSE;
		R3.FB_In.User_Inputs.6:= FALSE;
		R3.FB_In.User_Inputs.7:= FALSE;
			(*Configure Options Amounts*)
			R3.FB_In.Options.WeldCont_Amount:=0; 					(*Select amount of Spot Type Weld Controllers here (0 min, 4 max)*)
			R3.FB_In.Options.WaterStand_Amount:= 0;				(*Select amount of Water Stands here (0 min, 2 max)*)
			R3.FB_In.Options.MIGCont_Amount:= 1;					(*Select amount of MIG Type Weld Controllers here (0 min, 1 max)*)
			R3.FB_In.Options.Reamer_Amount:= 1;					(*Select amount of Tip Reamers here (0 min, 1 max)*)
			R3.FB_In.Options.EOAT_Amount:= 0;						(*Assign EOAT number to robot (0 min, 10 max)*)
			(*Configure Options Parameters*)
			
			R3.Reamer[1](
				(*FB Inputs*)
					Enable_Motion:= All_Estops_OK,
					Fronius_Ream:= TRUE,
                    Binzel_Ream:= FALSE,  (*optional*)
					
					Ream_REQ:= R3.Peripheral_Req.1 AND ((R3.Task_ID_Ack=Tip_Dress)OR (R3.In_T1 AND R3.Peripheral_Req.5)),
					Ream_Time:= T#2S,
					Ream_Clamp_Open:= R3.Reamer[1].N01.I.1,
					Spray_REQ:= R3.Peripheral_Req.2 AND ((R3.Task_ID_Ack=Tip_Dress)OR (R3.In_T1 AND R3.Peripheral_Req.5)),
					Spray_Time:= T#2S,
					F_WireCutter_REQ:= R3.Peripheral_Req.4 AND ((R3.Task_ID_Ack=Tip_Dress)OR (R3.In_T1 AND R3.Peripheral_Req.5)),
					F_WireCutter_Time:= T#1S,
					
				(*FB Outputs*)
					Reaming_Complete=> ,(*mapped in cell services*)
					(*The following are for Binzel type reamers only*)
					LifterUp_ACK=> , (*mapped in cell services*)
					Clamp_ACK=>,(*mapped in cell services*)
					Injector_ACK=> ,(*mapped in cell services*)
					WireCutter_ACK=> (*mapped in cell services*)
					);
			
			(*R3.Reamer[1](
				(*FB Inputs*)
					Enable_Motion:= All_Estops_OK,
					Fronius_Ream:= TRUE,
                    Binzel_Ream:= FALSE,  (*optional*)
					Ream_REQ:= R3.Peripheral_Req.5 AND (R3.Task_ID_Ack=Tip_Dress),

				(*FB Outputs*)
					Reaming_Complete=> ,(*mapped in cell services*)
					);*)
		(*Call Actual Object*)
		R3();
		(*Output Data*)
		Out_To_ICxx.Robot[3].Robot_Type:= R3.FB_In.Robot_Type;
		Out_To_ICxx.Robot[3].Status:= R3.Status;
		Out_To_ICxx.Robot[3].Axis_Data[1]:= R3.S_Axis_Pos_Raw;
		Out_To_ICxx.Robot[3].In_Image:= R3.Input_Image;
		Out_To_ICxx.Robot[3].Out_Image:= R3.Output_Image;
		Out_To_ICxx.Robot[3].Discrete_ImageFSOE:= R3.Discrete_Image_FSoE;
		Out_To_ICxx.Robot[3].Options:= R3.FB_In.Options;
			Out_To_ICxx.Robot[3].WS_Discrete_Image[1]:= R3.WS[1].Discrete_Image;
			Out_To_ICxx.Robot[3].WS_Discrete_Image[2]:= R3.WS[2].Discrete_Image;
 			Out_To_ICxx.Robot[3].ATI_Discrete_Image:= R3.ATI[1].Discrete_Image;
			Out_To_ICxx.Robot[3].Reamer_Discrete_Image:= R3.Reamer[1].Discrete_Image;
			Out_To_ICxx.Robot[3].Fronius_Status:= R3.Fronius_Status;
		Out_To_ICxx.Robot[3].Ped_IO_ToShow[1]:= 0;			(*Set to Ped value if this robots ecat string contains the Ped's IO*)
		Out_To_ICxx.Robot[3].Ped_IO_ToShow[2]:= 0;			(*Set to Ped value if this robots ecat string contains the Ped's IO*)
		Out_To_ICxx.Robot[3].ECAT_Cable_Breaks:= R3.ECatSlave_Cable_Breaks;
		Out_To_ICxx.Robot[3].CT:= R3.CT;


(*R4 ------------------------*)
		(*Input Data*)
		R4.FB_In.Robot_Type:=KUKA_KRC4_SAFEOP;
		R4.FB_In.Install_Zero_Orientation:= 0; 	(*Set this value between 0 and 359 to set the zero position of the robot physical install with reference to 12 o'clock symbol on UI screens*)
		R4.FB_In.Under_Construction:= GTAC_CONFIG.Under_Construction;
		R4.FB_In.In_SIM_Mode:= GTAC_CONFIG.In_SIM_Mode;
		R4.FB_In.SIM_StartWorkAround:= FALSE;  (*Main.SIM_WorkAround_StartRobots*)
		R4.FB_In.CoE_Read_Trigger:= (GTAC_CONFIG.Option_Robot_Count>=4) AND Pulse_CoERead;
		R4.FB_In.Ecat_Master_AmsNetID:= MAIN.ECAT_Master.AmsID;
		R4.FB_In.Prev_EcatNode_Present:= NOT R3.EK1100_NotPresent; (*Ensure Previous Node Exists to determine Ecat Cable Break of this Devices Input Cable*)
		R4.FB_In.Safety_RST:=SAFETY_RESET;
		R4.FB_In.Enable_Motion:= All_Estops_OK OR GTAC_CONFIG.Under_Construction;
		R4.FB_In.Alarm_RST:=In_From_ICxx.ControlPower1;
		R4.FB_In.Select_Play:=FALSE;
		R4.FB_In.Select_Teach:=FALSE;
		R4.FB_In.Select_Remote:=FALSE;
		R4.FB_In.Start_Scan:=In_From_ICxx.StartRobots;
		R4.FB_In.Stop_Scan:=In_From_ICxx.StopRobots;
		R4.FB_In.Stop_Scan2:=FALSE;
		R4.FB_In.In_DryCycle:= GTAC_CONFIG.Dry_Cycle_Enabled;
		R4.FB_In.Low_Speed:= GTAC_CONFIG.Low_Speed_Enabled;
		R4.FB_In.Speed_Request:= In_From_ICxx.Global_Robot_Speed;
		R4.FB_In.Force_MasterTest_Req:= Cell_Services_Prog.Human_Reqs_MasterTest OR Cell_Services_Prog.A_Robot_Reqs_MasterTest;
		R4.FB_In.Force_BrakeTest_Req:= Cell_Services_Prog.Human_Reqs_BrakeTest OR Cell_Services_Prog.A_Robot_Reqs_BrakeTest;
		R4.FB_In.Major_Faults:= Faults.System_Major_Fault;
		R4.FB_In.Teach_Interlock:=R4_Data.Teach_Interlock;
		R4.FB_In.Weld_Inhibit:=In_From_ICxx.Rxx_Weld_Inhibit;
		R4.FB_In.Option_Disable_WaterFLT:= FALSE AND GTAC_CONFIG.Under_Construction OR (MAIN.R4.Task_ID_Ack=Tip_Change_EXT); (*Used to disable water fault if no water is present. use with caution*)
		R4.FB_In.OK_ToEnter_EquipInterf1:=R4_Data.OK_ToEnter_EquipInterf1;
		R4.FB_In.OK_ToEnter_EquipInterf2:=R4_Data.OK_ToEnter_EquipInterf2;
		R4.FB_In.OK_ToEnter_EquipInterf3:=R4_Data.OK_ToEnter_EquipInterf3;
		R4.FB_In.OK_ToEnter_EquipInterf4:=R4_Data.OK_ToEnter_EquipInterf4;
		R4.FB_In.OK_ToEnter_EquipInterf5:=R4_Data.OK_ToEnter_EquipInterf5;
		R4.FB_In.OK_ToEnter_EquipInterf6:=R4_Data.OK_ToEnter_EquipInterf6;
		R4.FB_In.OK_ToEnter_EquipInterf7:=R4_Data.OK_ToEnter_EquipInterf7;
		R4.FB_In.OK_ToEnter_EquipInterf8:=R4_Data.OK_ToEnter_EquipInterf8;
		R4.FB_In.OK_ToEnter_EquipInterf9:=R4_Data.OK_ToEnter_EquipInterf9;
		R4.FB_In.OK_ToEnter_HumanInterf1:=R4_Data.OK_ToEnter_HumanInterf1;
		R4.FB_In.OK_ToEnter_HumanInterf2:=R4_Data.OK_ToEnter_HumanInterf2;
		R4.FB_In.OK_ToEnter_HumanInterf3:=R4_Data.OK_ToEnter_HumanInterf3;
		R4.FB_In.OK_ToEnter_HumanInterf4:=R4_Data.OK_ToEnter_HumanInterf4;
		R4.FB_In.OK_ToEnter_HumanInterf5:=R4_Data.OK_ToEnter_HumanInterf5;
		R4.FB_In.OK_ToEnter_HumanInterf6:=R4_Data.OK_ToEnter_HumanInterf6;
		R4.FB_In.OK_ToEnter_HumanInterf7:=R4_Data.OK_ToEnter_HumanInterf7;
		R4.FB_In.OK_ToEnter_RobotInterfs:= R4_Data.OK_ToEnter_RobotInterfs;
		R4.FB_In.Fix_ID:=R4_Data.Fix_ID[R4.Location_Index];
		R4.FB_In.Model_ID:=R4_Data.Model_ID[R4.Location_Index];
		R4.FB_In.Task_ID:=R4_Data.Task_ID[R4.Location_Index];
		R4.FB_In.Proceed_From_Pounce:=R4_Data.Proceed_From_Pounce[R4.Location_Index];
		R4.FB_In.Complete_Ack:=R4_Data.Complete_Ack[R4.Location_Index];
		R4.FB_In.PeripheralReq_Ack:=R4_Data.PeripheralReq_Ack[R4.Location_Index];
		R4.FB_In.AuxReq_Ack:=R4_Data.AuxReq_Ack[R4.Location_Index];
		R4.FB_In.User_Inputs.0:= FALSE;
		R4.FB_In.User_Inputs.1:= FALSE;
		R4.FB_In.User_Inputs.2:= FALSE;
		R4.FB_In.User_Inputs.3:= FALSE;
		R4.FB_In.User_Inputs.4:= FALSE;
		R4.FB_In.User_Inputs.5:= FALSE;
		R4.FB_In.User_Inputs.6:= FALSE;
		R4.FB_In.User_Inputs.7:= FALSE;
			(*Configure Options Amounts*)
			R4.FB_In.Options.WeldCont_Amount:=0; 					(*Select amount of Spot Type Weld Controllers here (0 min, 4 max)*)
			R4.FB_In.Options.WaterStand_Amount:= 0;				(*Select amount of Water Stands here (0 min, 2 max)*)
			R4.FB_In.Options.MIGCont_Amount:= 0;					(*Select amount of MIG Type Weld Controllers here (0 min, 1 max)*)
			R4.FB_In.Options.Reamer_Amount:= 0;					(*Select amount of Tip Reamers here (0 min, 1 max)*)
			R4.FB_In.Options.EOAT_Amount:= 1;						(*Assign EOAT number to robot (0 min, 10 max)*)
			(*Configure Options Parameters*)

		(*Call Actual Object*)
		R4();
		(*Output Data*)
		Out_To_ICxx.Robot[4].Robot_Type:= R4.FB_In.Robot_Type;
		Out_To_ICxx.Robot[4].Status:= R4.Status;
		Out_To_ICxx.Robot[4].Axis_Data[1]:= R4.S_Axis_Pos_Raw;
		Out_To_ICxx.Robot[4].Axis_Data[7]:= R4.External_Axis_Pos_Raw; (*Actual value coming from robot*)
		Out_To_ICxx.Robot[4].In_Image:= R4.Input_Image;
		Out_To_ICxx.Robot[4].Out_Image:= R4.Output_Image;
		Out_To_ICxx.Robot[4].Discrete_ImageFSOE:= R4.Discrete_Image_FSoE;
		Out_To_ICxx.Robot[4].Options:= R4.FB_In.Options;
			Out_To_ICxx.Robot[4].WS_Discrete_Image[1]:= R4.WS[1].Discrete_Image;
			Out_To_ICxx.Robot[4].WS_Discrete_Image[2]:= R4.WS[2].Discrete_Image;
 			Out_To_ICxx.Robot[4].ATI_Discrete_Image:= R4.ATI[1].Discrete_Image;
			Out_To_ICxx.Robot[4].Reamer_Discrete_Image:= R4.Reamer[1].Discrete_Image;
			Out_To_ICxx.Robot[4].Fronius_Status:= R4.Fronius_Status;
		Out_To_ICxx.Robot[4].Ped_IO_ToShow[1]:= 0;			(*Set to Ped value if this robots ecat string contains the Ped's IO*)
		Out_To_ICxx.Robot[4].Ped_IO_ToShow[2]:= 0;			(*Set to Ped value if this robots ecat string contains the Ped's IO*)
		Out_To_ICxx.Robot[4].ECAT_Cable_Breaks:= R4.ECatSlave_Cable_Breaks;
		Out_To_ICxx.Robot[4].CT:= R4.CT;



(*R5 ------------------------*)
		(*Input Data*)
		R5.FB_In.Robot_Type:=KUKA_KRC4_SAFEOP_Turntable;
		R5.FB_In.Install_Zero_Orientation:= 0; 	(*Set this value between 0 and 359 to set the zero position of the robot physical install with reference to 12 o'clock symbol on UI screens*)
		R5.FB_In.Under_Construction:= GTAC_CONFIG.Under_Construction;
		R5.FB_In.In_SIM_Mode:= GTAC_CONFIG.In_SIM_Mode;
		R5.FB_In.SIM_StartWorkAround:= FALSE;  (*Main.SIM_WorkAround_StartRobots*)
		R5.FB_In.CoE_Read_Trigger:= (GTAC_CONFIG.Option_Robot_Count>=5) AND Pulse_CoERead;
		R5.FB_In.Ecat_Master_AmsNetID:= MAIN.ECAT_Master.AmsID;
		R5.FB_In.Prev_EcatNode_Present:= NOT R4.EK1100_NotPresent; (*Ensure Previous Node Exists to determine Ecat Cable Break of this Devices Input Cable*)
		R5.FB_In.Safety_RST:=SAFETY_RESET;
		R5.FB_In.Enable_Motion:= All_Estops_OK OR GTAC_CONFIG.Under_Construction;
		R5.FB_In.Alarm_RST:=In_From_ICxx.ControlPower1;
		R5.FB_In.Select_Play:=FALSE;
		R5.FB_In.Select_Teach:=FALSE;
		R5.FB_In.Select_Remote:=FALSE;
		R5.FB_In.Start_Scan:=In_From_ICxx.StartRobots;
		R5.FB_In.Stop_Scan:=In_From_ICxx.StopRobots;
		R5.FB_In.Stop_Scan2:=FALSE;
		R5.FB_In.In_DryCycle:= GTAC_CONFIG.Dry_Cycle_Enabled;
		R5.FB_In.Low_Speed:= GTAC_CONFIG.Low_Speed_Enabled;
		R5.FB_In.Speed_Request:= In_From_ICxx.Global_Robot_Speed;
		R5.FB_In.Force_MasterTest_Req:= Cell_Services_Prog.Human_Reqs_MasterTest OR Cell_Services_Prog.A_Robot_Reqs_MasterTest;
		R5.FB_In.Force_BrakeTest_Req:= Cell_Services_Prog.Human_Reqs_BrakeTest OR Cell_Services_Prog.A_Robot_Reqs_BrakeTest;
		R5.FB_In.Major_Faults:= Faults.System_Major_Fault;
		R5.FB_In.Teach_Interlock:=R5_Data.Teach_Interlock;
		R5.FB_In.Weld_Inhibit:=In_From_ICxx.Rxx_Weld_Inhibit;
		R5.FB_In.Option_Disable_WaterFLT:= FALSE AND GTAC_CONFIG.Under_Construction OR (MAIN.R5.Task_ID_Ack=Tip_Change_EXT); (*Used to disable water fault if no water is present. use with caution*)
		R5.FB_In.OK_ToEnter_EquipInterf1:=R5_Data.OK_ToEnter_EquipInterf1;
		R5.FB_In.OK_ToEnter_EquipInterf2:=R5_Data.OK_ToEnter_EquipInterf2;
		R5.FB_In.OK_ToEnter_EquipInterf3:=R5_Data.OK_ToEnter_EquipInterf3;
		R5.FB_In.OK_ToEnter_EquipInterf4:=R5_Data.OK_ToEnter_EquipInterf4;
		R5.FB_In.OK_ToEnter_EquipInterf5:=R5_Data.OK_ToEnter_EquipInterf5;
		R5.FB_In.OK_ToEnter_EquipInterf6:=R5_Data.OK_ToEnter_EquipInterf6;
		R5.FB_In.OK_ToEnter_EquipInterf7:=R5_Data.OK_ToEnter_EquipInterf7;
		R5.FB_In.OK_ToEnter_EquipInterf8:=R5_Data.OK_ToEnter_EquipInterf8;
		R5.FB_In.OK_ToEnter_EquipInterf9:=R5_Data.OK_ToEnter_EquipInterf9;
		R5.FB_In.OK_ToEnter_HumanInterf1:=R5_Data.OK_ToEnter_HumanInterf1;
		R5.FB_In.OK_ToEnter_HumanInterf2:=R5_Data.OK_ToEnter_HumanInterf2;
		R5.FB_In.OK_ToEnter_HumanInterf3:=R5_Data.OK_ToEnter_HumanInterf3;
		R5.FB_In.OK_ToEnter_HumanInterf4:=R5_Data.OK_ToEnter_HumanInterf4;
		R5.FB_In.OK_ToEnter_HumanInterf5:=R5_Data.OK_ToEnter_HumanInterf5;
		R5.FB_In.OK_ToEnter_HumanInterf6:=R5_Data.OK_ToEnter_HumanInterf6;
		R5.FB_In.OK_ToEnter_HumanInterf7:=R5_Data.OK_ToEnter_HumanInterf7;
		R5.FB_In.OK_ToEnter_HumanInterf8:=R5_Data.OK_ToEnter_HumanInterf8;
		R5.FB_In.OK_ToEnter_RobotInterfs:= R5_Data.OK_ToEnter_RobotInterfs;
		R5.FB_In.Fix_ID:=R5_Data.Fix_ID[R5.Location_Index];
		R5.FB_In.Model_ID:=R5_Data.Model_ID[R5.Location_Index];
		R5.FB_In.Task_ID:=R5_Data.Task_ID[R5.Location_Index];
		R5.FB_In.Proceed_From_Pounce:=R5_Data.Proceed_From_Pounce[R5.Location_Index];
		R5.FB_In.Complete_Ack:=R5_Data.Complete_Ack[R5.Location_Index];
		R5.FB_In.PeripheralReq_Ack:=R5_Data.PeripheralReq_Ack[R5.Location_Index];
		R5.FB_In.AuxReq_Ack:=R5_Data.AuxReq_Ack[R5.Location_Index];
		R5.FB_In.User_Inputs.0:= FALSE;
		R5.FB_In.User_Inputs.1:= FALSE;
		R5.FB_In.User_Inputs.2:= FALSE;
		R5.FB_In.User_Inputs.3:= FALSE;
		R5.FB_In.User_Inputs.4:= FALSE;
		R5.FB_In.User_Inputs.5:= FALSE;
		R5.FB_In.User_Inputs.6:= FALSE;
		R5.FB_In.User_Inputs.7:= FALSE;
			(*Configure Options Amounts*)
			R5.FB_In.Options.WeldCont_Amount:= 0; 					(*Select amount of Spot Type Weld Controllers here (0 min, 4 max)*)
			R5.FB_In.Options.WaterStand_Amount:= 0;				(*Select amount of Water Stands here (0 min, 2 max)*)
			R5.FB_In.Options.MIGCont_Amount:= 1;					(*Select amount of MIG Type Weld Controllers here (0 min, 1 max)*)
			R5.FB_In.Options.Reamer_Amount:= 1;					(*Select amount of Tip Reamers here (0 min, 1 max)*)
			R5.FB_In.Options.EOAT_Amount:= 0;						(*Assign EOAT number to robot (0 min, 10 max)*)
			(*Configure Options Parameters*)
			
			R5.Reamer[1](
				(*FB Inputs*)
					Enable_Motion:= All_Estops_OK,
					Fronius_Ream:= TRUE,
                    Binzel_Ream:= FALSE,  (*optional*)
					
					Ream_REQ:= R5.Peripheral_Req.1 AND ((R5.Task_ID_Ack=Tip_Dress)OR (R5.In_T1 AND R5.Peripheral_Req.5)),
					Ream_Time:= T#2S,
					Ream_Clamp_Open:= R5.Reamer[1].N01.I.1,
					Spray_REQ:= R5.Peripheral_Req.2 AND ((R5.Task_ID_Ack=Tip_Dress)OR (R5.In_T1 AND R5.Peripheral_Req.5)),
					Spray_Time:= T#2S,
					F_WireCutter_REQ:= R5.Peripheral_Req.4 AND ((R5.Task_ID_Ack=Tip_Dress)OR (R5.In_T1 AND R5.Peripheral_Req.5)),
					F_WireCutter_Time:= T#1S,
					
				(*FB Outputs*)
					Reaming_Complete=> ,(*mapped in cell services*)
					(*The following are for Binzel type reamers only*)
					LifterUp_ACK=> , (*mapped in cell services*)
					Clamp_ACK=>,(*mapped in cell services*)
					Injector_ACK=> ,(*mapped in cell services*)
					WireCutter_ACK=> (*mapped in cell services*)
					);
			(*R5.Reamer[1](
				(*FB Inputs*)
					Enable_Motion:= All_Estops_OK,
					Fronius_Ream:= TRUE,
                    Binzel_Ream:= FALSE,  (*optional*)
					Ream_REQ:= R5.Peripheral_Req.5 AND (R5.Task_ID_Ack=Tip_Dress),

				(*FB Outputs*)
					Reaming_Complete=> ,(*mapped in cell services*)
					);*)
		(*Call Actual Object*)
		R5();
		(*Output Data*)
		Out_To_ICxx.Robot[5].Robot_Type:= R5.FB_In.Robot_Type;
		Out_To_ICxx.Robot[5].Status:= R5.Status;
		Out_To_ICxx.Robot[5].Axis_Data[1]:= R5.S_Axis_Pos_Raw;
		Out_To_ICxx.Robot[5].In_Image:= R5.Input_Image;
		Out_To_ICxx.Robot[5].Out_Image:= R5.Output_Image;
		Out_To_ICxx.Robot[5].Discrete_ImageFSOE:= R5.Discrete_Image_FSoE;
		Out_To_ICxx.Robot[5].Options:= R5.FB_In.Options;
			Out_To_ICxx.Robot[5].WS_Discrete_Image[1]:= R5.WS[1].Discrete_Image;
			Out_To_ICxx.Robot[5].WS_Discrete_Image[2]:= R5.WS[2].Discrete_Image;
 			Out_To_ICxx.Robot[5].ATI_Discrete_Image:= R5.ATI[1].Discrete_Image;
			Out_To_ICxx.Robot[5].Reamer_Discrete_Image:= R5.Reamer[1].Discrete_Image;
			Out_To_ICxx.Robot[5].Fronius_Status:= R5.Fronius_Status;
		Out_To_ICxx.Robot[5].Ped_IO_ToShow[1]:= 0;			(*Set to Ped value if this robots ecat string contains the Ped's IO*)
		Out_To_ICxx.Robot[5].Ped_IO_ToShow[2]:= 0;			(*Set to Ped value if this robots ecat string contains the Ped's IO*)
		Out_To_ICxx.Robot[5].ECAT_Cable_Breaks:= R5.ECatSlave_Cable_Breaks;
		Out_To_ICxx.Robot[5].CT:= R5.CT;
		(*Example of passing Turntable Axis Data*)
		//Out_To_ICxx.TT02_Location_Index:= R5.TT_Axis_Location_Index; (*Pass Turntable location*) DEBUG - RESTORE AFTER SIM - RJ
		
		(*IF (MAIN.SIM_WorkAround_TT02_Position_Index[0] = TRUE)
			THEN Out_To_ICxx.TT02_Location_Index:= 1;
		ELSIF (MAIN.SIM_WorkAround_TT02_Position_Index[1] = TRUE)
			THEN Out_To_ICxx.TT02_Location_Index:= 2;
		ELSE
			Out_To_ICxx.TT02_Location_Index:= 0;
		END_IF*)	//DEBUG - RJ - REMOVE ABOVE AFTER SIM, RESTORE original Out_To_ICxx.TT01_Location_Index:= R1.TT_Axis_Location_Index;
		Out_To_ICxx.TT02_Location_Index:= R5.TT_Axis_Location_Index;



(*R6 ------------------------*)
		(*Input Data*)
		R6.FB_In.Robot_Type:=KUKA_KRC4_SAFEOP;
		R6.FB_In.Install_Zero_Orientation:= 0; 	(*Set this value between 0 and 359 to set the zero position of the robot physical install with reference to 12 o'clock symbol on UI screens*)
		R6.FB_In.Under_Construction:= GTAC_CONFIG.Under_Construction;
		R6.FB_In.In_SIM_Mode:= GTAC_CONFIG.In_SIM_Mode;
		R6.FB_In.SIM_StartWorkAround:= FALSE;  (*Main.SIM_WorkAround_StartRobots*)
		R6.FB_In.CoE_Read_Trigger:= (GTAC_CONFIG.Option_Robot_Count>=6) AND Pulse_CoERead;
		R6.FB_In.Ecat_Master_AmsNetID:= MAIN.ECAT_Master.AmsID;
		R6.FB_In.Prev_EcatNode_Present:= NOT R5.EK1100_NotPresent; (*Ensure Previous Node Exists to determine Ecat Cable Break of this Devices Input Cable*)
		R6.FB_In.Safety_RST:=SAFETY_RESET;
		R6.FB_In.Enable_Motion:= All_Estops_OK OR GTAC_CONFIG.Under_Construction;
		R6.FB_In.Alarm_RST:=In_From_ICxx.ControlPower1;
		R6.FB_In.Select_Play:=FALSE;
		R6.FB_In.Select_Teach:=FALSE;
		R6.FB_In.Select_Remote:=FALSE;
		R6.FB_In.Start_Scan:=In_From_ICxx.StartRobots;
		R6.FB_In.Stop_Scan:=In_From_ICxx.StopRobots;
		R6.FB_In.Stop_Scan2:=FALSE;
		R6.FB_In.In_DryCycle:= GTAC_CONFIG.Dry_Cycle_Enabled;
		R6.FB_In.Low_Speed:= GTAC_CONFIG.Low_Speed_Enabled;
		R6.FB_In.Speed_Request:= In_From_ICxx.Global_Robot_Speed;
		R6.FB_In.Force_MasterTest_Req:= Cell_Services_Prog.Human_Reqs_MasterTest OR Cell_Services_Prog.A_Robot_Reqs_MasterTest;
		R6.FB_In.Force_BrakeTest_Req:= Cell_Services_Prog.Human_Reqs_BrakeTest OR Cell_Services_Prog.A_Robot_Reqs_BrakeTest;
		R6.FB_In.Major_Faults:= Faults.System_Major_Fault;
		R6.FB_In.Teach_Interlock:=R6_Data.Teach_Interlock;
		R6.FB_In.Weld_Inhibit:=In_From_ICxx.Rxx_Weld_Inhibit;
		R6.FB_In.Option_Disable_WaterFLT:= FALSE AND GTAC_CONFIG.Under_Construction OR (MAIN.R6.Task_ID_Ack=Tip_Change_EXT); (*Used to disable water fault if no water is present. use with caution*)
		R6.FB_In.OK_ToEnter_EquipInterf1:=R6_Data.OK_ToEnter_EquipInterf1;
		R6.FB_In.OK_ToEnter_EquipInterf2:=R6_Data.OK_ToEnter_EquipInterf2;
		R6.FB_In.OK_ToEnter_EquipInterf3:=R6_Data.OK_ToEnter_EquipInterf3;
		R6.FB_In.OK_ToEnter_EquipInterf4:=R6_Data.OK_ToEnter_EquipInterf4;
		R6.FB_In.OK_ToEnter_EquipInterf5:=R6_Data.OK_ToEnter_EquipInterf5;
		R6.FB_In.OK_ToEnter_EquipInterf6:=R6_Data.OK_ToEnter_EquipInterf6;
		R6.FB_In.OK_ToEnter_EquipInterf7:=R6_Data.OK_ToEnter_EquipInterf7;
		R6.FB_In.OK_ToEnter_EquipInterf8:=R6_Data.OK_ToEnter_EquipInterf8;
		R6.FB_In.OK_ToEnter_EquipInterf9:=R6_Data.OK_ToEnter_EquipInterf9;
		R6.FB_In.OK_ToEnter_HumanInterf1:=R6_Data.OK_ToEnter_HumanInterf1;
		R6.FB_In.OK_ToEnter_HumanInterf2:=R6_Data.OK_ToEnter_HumanInterf2;
		R6.FB_In.OK_ToEnter_HumanInterf3:=R6_Data.OK_ToEnter_HumanInterf3;
		R6.FB_In.OK_ToEnter_HumanInterf4:=R6_Data.OK_ToEnter_HumanInterf4;
		R6.FB_In.OK_ToEnter_HumanInterf5:=R6_Data.OK_ToEnter_HumanInterf5;
		R6.FB_In.OK_ToEnter_HumanInterf6:=R6_Data.OK_ToEnter_HumanInterf6;
		R6.FB_In.OK_ToEnter_HumanInterf7:=R6_Data.OK_ToEnter_HumanInterf7;
		R6.FB_In.OK_ToEnter_HumanInterf8:=R6_Data.OK_ToEnter_HumanInterf8;
		R6.FB_In.OK_ToEnter_RobotInterfs:= R6_Data.OK_ToEnter_RobotInterfs;
		R6.FB_In.Fix_ID:=R6_Data.Fix_ID[R6.Location_Index];
		R6.FB_In.Model_ID:=R6_Data.Model_ID[R6.Location_Index];
		R6.FB_In.Task_ID:=R6_Data.Task_ID[R6.Location_Index];
		R6.FB_In.Proceed_From_Pounce:=R6_Data.Proceed_From_Pounce[R6.Location_Index];
		R6.FB_In.Complete_Ack:=R6_Data.Complete_Ack[R6.Location_Index];
		R6.FB_In.PeripheralReq_Ack:=R6_Data.PeripheralReq_Ack[R6.Location_Index];
		R6.FB_In.AuxReq_Ack:=R6_Data.AuxReq_Ack[R6.Location_Index];
		R6.FB_In.User_Inputs.0:= FALSE;
		R6.FB_In.User_Inputs.1:= FALSE;
		R6.FB_In.User_Inputs.2:= FALSE;
		R6.FB_In.User_Inputs.3:= FALSE;
		R6.FB_In.User_Inputs.4:= FALSE;
		R6.FB_In.User_Inputs.5:= FALSE;
		R6.FB_In.User_Inputs.6:= FALSE;
		R6.FB_In.User_Inputs.7:= FALSE;
			(*Configure Options Amounts*)
			R6.FB_In.Options.WeldCont_Amount:= 0; 					(*Select amount of Spot Type Weld Controllers here (0 min, 4 max)*)
			R6.FB_In.Options.WaterStand_Amount:= 0;				(*Select amount of Water Stands here (0 min, 2 max)*)
			R6.FB_In.Options.MIGCont_Amount:= 1;					(*Select amount of MIG Type Weld Controllers here (0 min, 1 max)*)
			R6.FB_In.Options.Reamer_Amount:= 1;					(*Select amount of Tip Reamers here (0 min, 1 max)*)
			R6.FB_In.Options.EOAT_Amount:= 0;						(*Assign EOAT number to robot (0 min, 10 max)*)
			(*Configure Options Parameters*)
			
			R6.Reamer[1](
				(*FB Inputs*)
					Enable_Motion:= All_Estops_OK,
					Fronius_Ream:= TRUE,
                    Binzel_Ream:= FALSE,  (*optional*)
					
					Ream_REQ:= R6.Peripheral_Req.1 AND ((R6.Task_ID_Ack=Tip_Dress)OR (R6.In_T1 AND R6.Peripheral_Req.5)),
					Ream_Time:= T#2S,
					Ream_Clamp_Open:= R6.Reamer[1].N01.I.1,
					Spray_REQ:= R6.Peripheral_Req.2 AND ((R6.Task_ID_Ack=Tip_Dress)OR (R6.In_T1 AND R6.Peripheral_Req.5)),
					Spray_Time:= T#2S,
					F_WireCutter_REQ:= R6.Peripheral_Req.4 AND ((R6.Task_ID_Ack=Tip_Dress)OR (R6.In_T1 AND R6.Peripheral_Req.5)),
					F_WireCutter_Time:= T#1S,
					
				(*FB Outputs*)
					Reaming_Complete=> ,(*mapped in cell services*)
					(*The following are for Binzel type reamers only*)
					LifterUp_ACK=> , (*mapped in cell services*)
					Clamp_ACK=>,(*mapped in cell services*)
					Injector_ACK=> ,(*mapped in cell services*)
					WireCutter_ACK=> (*mapped in cell services*)
					);
			(*R6.Reamer[1](
				(*FB Inputs*)
					Enable_Motion:= All_Estops_OK,
					Fronius_Ream:= TRUE,
                    Binzel_Ream:= FALSE,  (*optional*)
					Ream_REQ:= R6.Peripheral_Req.5 AND (R6.Task_ID_Ack=Tip_Dress),

				(*FB Outputs*)
					Reaming_Complete=> ,(*mapped in cell services*)
					);*)
		(*Call Actual Object*)
		R6();
		(*Output Data*)
		Out_To_ICxx.Robot[6].Robot_Type:= R6.FB_In.Robot_Type;
		Out_To_ICxx.Robot[6].Status:= R6.Status;
		Out_To_ICxx.Robot[6].Axis_Data[1]:= R6.S_Axis_Pos_Raw;
		Out_To_ICxx.Robot[6].In_Image:= R6.Input_Image;
		Out_To_ICxx.Robot[6].Out_Image:= R6.Output_Image;
		Out_To_ICxx.Robot[6].Discrete_ImageFSOE:= R6.Discrete_Image_FSoE;
		Out_To_ICxx.Robot[6].Options:= R6.FB_In.Options;
			Out_To_ICxx.Robot[6].WS_Discrete_Image[1]:= R6.WS[1].Discrete_Image;
			Out_To_ICxx.Robot[6].WS_Discrete_Image[2]:= R6.WS[2].Discrete_Image;
 			Out_To_ICxx.Robot[6].ATI_Discrete_Image:= R6.ATI[1].Discrete_Image;
			Out_To_ICxx.Robot[6].Reamer_Discrete_Image:= R6.Reamer[1].Discrete_Image;
			Out_To_ICxx.Robot[6].Fronius_Status:= R6.Fronius_Status;
		Out_To_ICxx.Robot[6].Ped_IO_ToShow[1]:= 0;			(*Set to Ped value if this robots ecat string contains the Ped's IO*)
		Out_To_ICxx.Robot[6].Ped_IO_ToShow[2]:= 0;			(*Set to Ped value if this robots ecat string contains the Ped's IO*)
		Out_To_ICxx.Robot[6].ECAT_Cable_Breaks:= R6.ECatSlave_Cable_Breaks;
		Out_To_ICxx.Robot[6].CT:= R6.CT;



(*R7 ------------------------*)
		(*Input Data*)
		R7.FB_In.Robot_Type:=KUKA_KRC4_SAFEOP;
		R7.FB_In.Install_Zero_Orientation:= 0; 	(*Set this value between 0 and 359 to set the zero position of the robot physical install with reference to 12 o'clock symbol on UI screens*)
		R7.FB_In.Under_Construction:= GTAC_CONFIG.Under_Construction;
		R7.FB_In.In_SIM_Mode:= GTAC_CONFIG.In_SIM_Mode;
		R7.FB_In.SIM_StartWorkAround:= FALSE;  (*Main.SIM_WorkAround_StartRobots*)
		R7.FB_In.CoE_Read_Trigger:= (GTAC_CONFIG.Option_Robot_Count>=7) AND Pulse_CoERead;
		R7.FB_In.Ecat_Master_AmsNetID:= MAIN.ECAT_Master.AmsID;
		R7.FB_In.Prev_EcatNode_Present:= NOT R6.EK1100_NotPresent; (*Ensure Previous Node Exists to determine Ecat Cable Break of this Devices Input Cable*)
		R7.FB_In.Safety_RST:=SAFETY_RESET;
		R7.FB_In.Enable_Motion:= All_Estops_OK OR GTAC_CONFIG.Under_Construction;
		R7.FB_In.Alarm_RST:=In_From_ICxx.ControlPower1;
		R7.FB_In.Select_Play:=FALSE;
		R7.FB_In.Select_Teach:=FALSE;
		R7.FB_In.Select_Remote:=FALSE;
		R7.FB_In.Start_Scan:=In_From_ICxx.StartRobots;
		R7.FB_In.Stop_Scan:=In_From_ICxx.StopRobots;
		R7.FB_In.Stop_Scan2:=FALSE;
		R7.FB_In.In_DryCycle:= GTAC_CONFIG.Dry_Cycle_Enabled;
		R7.FB_In.Low_Speed:= GTAC_CONFIG.Low_Speed_Enabled;
		R7.FB_In.Speed_Request:= In_From_ICxx.Global_Robot_Speed;
		R7.FB_In.Force_MasterTest_Req:= Cell_Services_Prog.Human_Reqs_MasterTest OR Cell_Services_Prog.A_Robot_Reqs_MasterTest;
		R7.FB_In.Force_BrakeTest_Req:= Cell_Services_Prog.Human_Reqs_BrakeTest OR Cell_Services_Prog.A_Robot_Reqs_BrakeTest;
		R7.FB_In.Major_Faults:= Faults.System_Major_Fault;
		R7.FB_In.Teach_Interlock:=R7_Data.Teach_Interlock;
		R7.FB_In.Weld_Inhibit:=In_From_ICxx.Rxx_Weld_Inhibit;
		R7.FB_In.Option_Disable_WaterFLT:= FALSE AND GTAC_CONFIG.Under_Construction OR (MAIN.R7.Task_ID_Ack=Tip_Change_EXT); (*Used to disable water fault if no water is present. use with caution*)
		R7.FB_In.OK_ToEnter_EquipInterf1:=R7_Data.OK_ToEnter_EquipInterf1;
		R7.FB_In.OK_ToEnter_EquipInterf2:=R7_Data.OK_ToEnter_EquipInterf2;
		R7.FB_In.OK_ToEnter_EquipInterf3:=R7_Data.OK_ToEnter_EquipInterf3;
		R7.FB_In.OK_ToEnter_EquipInterf4:=R7_Data.OK_ToEnter_EquipInterf4;
		R7.FB_In.OK_ToEnter_EquipInterf5:=R7_Data.OK_ToEnter_EquipInterf5;
		R7.FB_In.OK_ToEnter_EquipInterf6:=R7_Data.OK_ToEnter_EquipInterf6;
		R7.FB_In.OK_ToEnter_EquipInterf7:=R7_Data.OK_ToEnter_EquipInterf7;
		R7.FB_In.OK_ToEnter_EquipInterf8:=R7_Data.OK_ToEnter_EquipInterf8;
		R7.FB_In.OK_ToEnter_EquipInterf9:=R7_Data.OK_ToEnter_EquipInterf9;
		R7.FB_In.OK_ToEnter_HumanInterf1:=R7_Data.OK_ToEnter_HumanInterf1;
		R7.FB_In.OK_ToEnter_HumanInterf2:=R7_Data.OK_ToEnter_HumanInterf2;
		R7.FB_In.OK_ToEnter_HumanInterf3:=R7_Data.OK_ToEnter_HumanInterf3;
		R7.FB_In.OK_ToEnter_HumanInterf4:=R7_Data.OK_ToEnter_HumanInterf4;
		R7.FB_In.OK_ToEnter_HumanInterf5:=R7_Data.OK_ToEnter_HumanInterf5;
		R7.FB_In.OK_ToEnter_HumanInterf6:=R7_Data.OK_ToEnter_HumanInterf6;
		R7.FB_In.OK_ToEnter_HumanInterf7:=R7_Data.OK_ToEnter_HumanInterf7;
		R7.FB_In.OK_ToEnter_HumanInterf8:=R7_Data.OK_ToEnter_HumanInterf8;
		R7.FB_In.OK_ToEnter_RobotInterfs:= R7_Data.OK_ToEnter_RobotInterfs;
		R7.FB_In.Fix_ID:=R7_Data.Fix_ID[R7.Location_Index];
		R7.FB_In.Model_ID:=R7_Data.Model_ID[R7.Location_Index];
		R7.FB_In.Task_ID:=R7_Data.Task_ID[R7.Location_Index];
		R7.FB_In.Proceed_From_Pounce:=R7_Data.Proceed_From_Pounce[R7.Location_Index];
		R7.FB_In.Complete_Ack:=R7_Data.Complete_Ack[R7.Location_Index];
		R7.FB_In.PeripheralReq_Ack:=R7_Data.PeripheralReq_Ack[R7.Location_Index];
		R7.FB_In.AuxReq_Ack:=R7_Data.AuxReq_Ack[R7.Location_Index];
		R7.FB_In.User_Inputs.0:= FALSE;
		R7.FB_In.User_Inputs.1:= FALSE;
		R7.FB_In.User_Inputs.2:= FALSE;
		R7.FB_In.User_Inputs.3:= FALSE;
		R7.FB_In.User_Inputs.4:= FALSE;
		R7.FB_In.User_Inputs.5:= FALSE;
		R7.FB_In.User_Inputs.6:= FALSE;
		R7.FB_In.User_Inputs.7:= FALSE;
			(*Configure Options Amounts*)
			R7.FB_In.Options.WeldCont_Amount:= 0; 					(*Select amount of Spot Type Weld Controllers here (0 min, 4 max)*)
			R7.FB_In.Options.WaterStand_Amount:= 0;				(*Select amount of Water Stands here (0 min, 2 max)*)
			R7.FB_In.Options.MIGCont_Amount:= 1;					(*Select amount of MIG Type Weld Controllers here (0 min, 1 max)*)
			R7.FB_In.Options.Reamer_Amount:= 1;					(*Select amount of Tip Reamers here (0 min, 1 max)*)
			R7.FB_In.Options.EOAT_Amount:= 0;						(*Assign EOAT number to robot (0 min, 10 max)*)
			(*Configure Options Parameters*)
			
			R7.Reamer[1](
				(*FB Inputs*)
					Enable_Motion:= All_Estops_OK,
					Fronius_Ream:= TRUE,
                    Binzel_Ream:= FALSE,  (*optional*)
					
					Ream_REQ:= R7.Peripheral_Req.1 AND ((R7.Task_ID_Ack=Tip_Dress)OR (R7.In_T1 AND R7.Peripheral_Req.5)),
					Ream_Time:= T#2S,
					Ream_Clamp_Open:= R7.Reamer[1].N01.I.1,
					Spray_REQ:= R7.Peripheral_Req.2 AND ((R7.Task_ID_Ack=Tip_Dress)OR (R7.In_T1 AND R7.Peripheral_Req.5)),
					Spray_Time:= T#2S,
					F_WireCutter_REQ:= R7.Peripheral_Req.4 AND ((R7.Task_ID_Ack=Tip_Dress)OR (R7.In_T1 AND R7.Peripheral_Req.5)),
					F_WireCutter_Time:= T#1S,
					
				(*FB Outputs*)
					Reaming_Complete=> ,(*mapped in cell services*)
					(*The following are for Binzel type reamers only*)
					LifterUp_ACK=> , (*mapped in cell services*)
					Clamp_ACK=>,(*mapped in cell services*)
					Injector_ACK=> ,(*mapped in cell services*)
					WireCutter_ACK=> (*mapped in cell services*)
					);
			(*R7.Reamer[1](
				(*FB Inputs*)
					Enable_Motion:= All_Estops_OK,
					Fronius_Ream:= TRUE,
                    Binzel_Ream:= FALSE,  (*optional*)
					Ream_REQ:= R7.Peripheral_Req.5 AND (R7.Task_ID_Ack=Tip_Dress),

				(*FB Outputs*)
					Reaming_Complete=> ,(*mapped in cell services*)
					);*)
		(*Call Actual Object*)
		R7();
		(*Output Data*)
		Out_To_ICxx.Robot[7].Robot_Type:= R7.FB_In.Robot_Type;
		Out_To_ICxx.Robot[7].Status:= R7.Status;
		Out_To_ICxx.Robot[7].Axis_Data[1]:= R7.S_Axis_Pos_Raw;
		Out_To_ICxx.Robot[7].In_Image:= R7.Input_Image;
		Out_To_ICxx.Robot[7].Out_Image:= R7.Output_Image;
		Out_To_ICxx.Robot[7].Discrete_ImageFSOE:= R7.Discrete_Image_FSoE;
		Out_To_ICxx.Robot[7].Options:= R7.FB_In.Options;
			Out_To_ICxx.Robot[7].WS_Discrete_Image[1]:= R7.WS[1].Discrete_Image;
			Out_To_ICxx.Robot[7].WS_Discrete_Image[2]:= R7.WS[2].Discrete_Image;
 			Out_To_ICxx.Robot[7].ATI_Discrete_Image:= R7.ATI[1].Discrete_Image;
			Out_To_ICxx.Robot[7].Reamer_Discrete_Image:= R7.Reamer[1].Discrete_Image;
			Out_To_ICxx.Robot[7].Fronius_Status:= R7.Fronius_Status;
		Out_To_ICxx.Robot[7].Ped_IO_ToShow[1]:= 0;			(*Set to Ped value if this robots ecat string contains the Ped's IO*)
		Out_To_ICxx.Robot[7].Ped_IO_ToShow[2]:= 0;			(*Set to Ped value if this robots ecat string contains the Ped's IO*)
		Out_To_ICxx.Robot[7].ECAT_Cable_Breaks:= R7.ECatSlave_Cable_Breaks;
		Out_To_ICxx.Robot[7].CT:= R7.CT;



